(* Logix 5000 project; controller Comas_L4 vendor 1 type 14 code 193 rev 30.11; software revision 30.02; part 5 of 12 *)

VAR_GLOBAL   (* controller tags *)
   Activation_Mode_Once : BOOL;
   Activation_Pompe : BOOL := 1;
   Activation_Rouleau : BOOL := 1;
   Activation_Synchro_Directe_Codeur : BOOL := 1;
   AOI_Badge : Badges_Acces := (Tempo_Logout_1 := 600000, Tempo_Logout_2 := 3600000, Tempo_Logout_3 := 3600000);
   AOI_Cam_Display_Horiz : AOI_CamDisplay_OCX_StdCAM := (Sts_EN := 1);
   AOI_Cam_Display_Verti : AOI_CamDisplay_OCX_StdCAM := (Sts_EN := 1);
   AOI_Pilotage_Codeur_Vitesse_Moy : Pilotage_Vitesse_Rapide_V4 := (Vitesse := 46.548676, Acc := 1000.0, Dec := 1000.0, Jerk := 25.0, Autorisation := 1, St_Vitesse := 1);
   Axe_Codeur_Four : AXIS_CIP_DRIVE;
   Axe_Comas : MOTION_GROUP;
   Axe_Coupe_Fil : AXIS_CIP_DRIVE;
   Axe_Horizontal_Droit : AXIS_CIP_DRIVE;
   Axe_Horizontal_Gauche : AXIS_CIP_DRIVE;
   Axe_Pompe_Doseuse : AXIS_CIP_DRIVE;
   Axe_Rouleaux_Canneles : AXIS_CIP_DRIVE;
   Axe_Vertical_Droit : AXIS_CIP_DRIVE;
   Axe_Vertical_Gauche : AXIS_CIP_DRIVE;
   Axe_Virtuel_Codeur : AXIS_VIRTUAL;
   Axe_Virtuel_Codeur_test : AXIS_VIRTUAL;
   Axe_Virtuel_Coupe_Fil : AXIS_VIRTUAL;
   Axe_Virtuel_Maitre : AXIS_VIRTUAL;
   Badge_Code_A : BOOL;
   Badge_Code_B : BOOL;
   Badge_Code_C : BOOL;
   Badge_Code_D : BOOL;
   BP_O_F_Trappe : BOOL;
   Cadencement_Moyennage_Codeur : FBD_TIMER := (TimerEnable := 1, PRE := 1000, ACC := 930, EN := 1, TT := 1);
   Cam_Chart_Horiz : Chart := (NumberOfDataPoints := 130, X_Axis_Min := -1.0, X_Axis_Max := 90.0, Y_Axis_Min := -52.012157, Y_Axis_Max := 87.0, DataSeries_FixedAxis.Visible := 1, DataSeries_FixedAxis.Data[1] := 0.6923077, DataSeries_FixedAxis.Data[2] := 1.3846154, DataSeries_FixedAxis.Data[3] := 2.0769231, DataSeries_FixedAxis.Data[4] := 2.7692308, DataSeries_FixedAxis.Data[5] := 3.4615386, DataSeries_FixedAxis.Data[6] := 4.1538463, DataSeries_FixedAxis.Data[7] := 4.846154, DataSeries_FixedAxis.Data[8] := 5.5384617, DataSeries_FixedAxis.Data[9] := 6.230769, DataSeries_FixedAxis.Data[10] := 6.9230766, DataSeries_FixedAxis.Data[11] := 7.615384, DataSeries_FixedAxis.Data[12] := 8.307692, DataSeries_FixedAxis.Data[13] := 8.999999, DataSeries_FixedAxis.Data[14] := 9.6923065, DataSeries_FixedAxis.Data[15] := 10.384614, DataSeries_FixedAxis.Data[16] := 11.076921, DataSeries_FixedAxis.Data[17] := 11.769229, DataSeries_FixedAxis.Data[18] := 12.461536, DataSeries_FixedAxis.Data[19] := 13.153844, DataSeries_FixedAxis.Data[20] := 13.846151, DataSeries_FixedAxis.Data[21] := 14.538459, DataSeries_FixedAxis.Data[22] := 15.230766, DataSeries_FixedAxis.Data[23] := 15.923074, DataSeries_FixedAxis.Data[24] := 16.615381, DataSeries_FixedAxis.Data[25] := 17.30769, DataSeries_FixedAxis.Data[26] := 17.999998, DataSeries_FixedAxis.Data[27] := 18.692307, DataSeries_FixedAxis.Data[28] := 19.384615, DataSeries_FixedAxis.Data[29] := 20.076923, DataSeries_FixedAxis.Data[30] := 20.769232, DataSeries_FixedAxis.Data[31] := 21.46154, DataSeries_FixedAxis.Data[32] := 22.153849, DataSeries_FixedAxis.Data[33] := 22.846157, DataSeries_FixedAxis.Data[34] := 23.538465, DataSeries_FixedAxis.Data[35] := 24.230774, DataSeries_FixedAxis.Data[36] := 24.923082, DataSeries_FixedAxis.Data[37] := 25.61539, DataSeries_FixedAxis.Data[38] := 26.3077, DataSeries_FixedAxis.Data[39] := 27.000008, DataSeries_FixedAxis.Data[40] := 27.692316, DataSeries_FixedAxis.Data[41] := 28.384624, DataSeries_FixedAxis.Data[42] := 29.076933, DataSeries_FixedAxis.Data[43] := 29.769241, DataSeries_FixedAxis.Data[44] := 30.46155, DataSeries_FixedAxis.Data[45] := 31.153858, DataSeries_FixedAxis.Data[46] := 31.846167, DataSeries_FixedAxis.Data[47] := 32.538475, DataSeries_FixedAxis.Data[48] := 33.23078, DataSeries_FixedAxis.Data[49] := 33.923088, DataSeries_FixedAxis.Data[50] := 34.615395, DataSeries_FixedAxis.Data[51] := 35.3077, DataSeries_FixedAxis.Data[52] := 36.000008, DataSeries_FixedAxis.Data[53] := 36.692314, DataSeries_FixedAxis.Data[54] := 37.38462,
        DataSeries_FixedAxis.Data[55] := 38.076927, DataSeries_FixedAxis.Data[56] := 38.769234, DataSeries_FixedAxis.Data[57] := 39.46154, DataSeries_FixedAxis.Data[58] := 40.153847, DataSeries_FixedAxis.Data[59] := 40.846153, DataSeries_FixedAxis.Data[60] := 41.53846, DataSeries_FixedAxis.Data[61] := 42.230766, DataSeries_FixedAxis.Data[62] := 42.923073, DataSeries_FixedAxis.Data[63] := 43.61538, DataSeries_FixedAxis.Data[64] := 44.307686, DataSeries_FixedAxis.Data[65] := 44.999992, DataSeries_FixedAxis.Data[66] := 45.6923, DataSeries_FixedAxis.Data[67] := 46.384605, DataSeries_FixedAxis.Data[68] := 47.076912, DataSeries_FixedAxis.Data[69] := 47.76922, DataSeries_FixedAxis.Data[70] := 48.461525, DataSeries_FixedAxis.Data[71] := 49.15383, DataSeries_FixedAxis.Data[72] := 49.846138, DataSeries_FixedAxis.Data[73] := 50.538445, DataSeries_FixedAxis.Data[74] := 51.23075, DataSeries_FixedAxis.Data[75] := 51.923058, DataSeries_FixedAxis.Data[76] := 52.615364, DataSeries_FixedAxis.Data[77] := 53.30767, DataSeries_FixedAxis.Data[78] := 53.999977, DataSeries_FixedAxis.Data[79] := 54.692284, DataSeries_FixedAxis.Data[80] := 55.38459, DataSeries_FixedAxis.Data[81] := 56.076897, DataSeries_FixedAxis.Data[82] := 56.769203, DataSeries_FixedAxis.Data[83] := 57.46151, DataSeries_FixedAxis.Data[84] := 58.153816, DataSeries_FixedAxis.Data[85] := 58.846123, DataSeries_FixedAxis.Data[86] := 59.53843, DataSeries_FixedAxis.Data[87] := 60.230736, DataSeries_FixedAxis.Data[88] := 60.923042, DataSeries_FixedAxis.Data[89] := 61.61535, DataSeries_FixedAxis.Data[90] := 62.307655, DataSeries_FixedAxis.Data[91] := 62.99996, DataSeries_FixedAxis.Data[92] := 63.69227, DataSeries_FixedAxis.Data[93] := 64.384575, DataSeries_FixedAxis.Data[94] := 65.07688, DataSeries_FixedAxis.Data[95] := 65.76919, DataSeries_FixedAxis.Data[96] := 66.461494, DataSeries_FixedAxis.Data[97] := 67.1538, DataSeries_FixedAxis.Data[98] := 67.84611, DataSeries_FixedAxis.Data[99] := 68.538414, DataSeries_FixedAxis.Data[100] := 69.23072, DataSeries_FixedAxis.Data[101] := 69.92303, DataSeries_FixedAxis.Data[102] := 70.61533, DataSeries_FixedAxis.Data[103] := 71.30764, DataSeries_FixedAxis.Data[104] := 71.99995, DataSeries_FixedAxis.Data[105] := 72.69225, DataSeries_FixedAxis.Data[106] := 73.38456, DataSeries_FixedAxis.Data[107] := 74.076866, DataSeries_FixedAxis.Data[108] := 74.76917, DataSeries_FixedAxis.Data[109] := 75.46148, DataSeries_FixedAxis.Data[110] := 76.153786, DataSeries_FixedAxis.Data[111] := 76.84609, DataSeries_FixedAxis.Data[112] := 77.5384, DataSeries_FixedAxis.Data[113] := 78.230705, DataSeries_FixedAxis.Data[114] := 78.92301,
        DataSeries_FixedAxis.Data[115] := 79.61532, DataSeries_FixedAxis.Data[116] := 80.307625, DataSeries_FixedAxis.Data[117] := 80.99993, DataSeries_FixedAxis.Data[118] := 81.69224, DataSeries_FixedAxis.Data[119] := 82.384544, DataSeries_FixedAxis.Data[120] := 83.07685, DataSeries_FixedAxis.Data[121] := 83.76916, DataSeries_FixedAxis.Data[122] := 84.461464, DataSeries_FixedAxis.Data[123] := 85.15377, DataSeries_FixedAxis.Data[124] := 85.84608, DataSeries_FixedAxis.Data[125] := 86.53838, DataSeries_FixedAxis.Data[126] := 87.23069, DataSeries_FixedAxis.Data[127] := 87.923, DataSeries_FixedAxis.Data[128] := 88.6153, DataSeries_FixedAxis.Data[129] := 90.0, DataSeries_1.Label := 'Position', DataSeries_1.Visible := 1, DataSeries_1.Data[2] := 0.018661816, DataSeries_1.Data[3] := 0.15915523, DataSeries_1.Data[4] := 0.46422943, DataSeries_1.Data[5] := 0.96573883, DataSeries_1.Data[6] := 1.6955377, DataSeries_1.Data[7] := 2.6854808, DataSeries_1.Data[8] := 3.9674213, DataSeries_1.Data[9] := 5.553846, DataSeries_1.Data[10] := 7.215384, DataSeries_1.Data[11] := 8.876922, DataSeries_1.Data[12] := 10.53846, DataSeries_1.Data[13] := 12.199998, DataSeries_1.Data[14] := 13.861536, DataSeries_1.Data[15] := 15.523073, DataSeries_1.Data[16] := 17.184612, DataSeries_1.Data[17] := 18.84615, DataSeries_1.Data[18] := 20.507687, DataSeries_1.Data[19] := 22.169226, DataSeries_1.Data[20] := 23.830763, DataSeries_1.Data[21] := 25.492302, DataSeries_1.Data[22] := 27.15384, DataSeries_1.Data[23] := 28.815376, DataSeries_1.Data[24] := 30.476915, DataSeries_1.Data[25] := 32.138454, DataSeries_1.Data[26] := 33.799995, DataSeries_1.Data[27] := 35.461536, DataSeries_1.Data[28] := 37.123077, DataSeries_1.Data[29] := 38.784615, DataSeries_1.Data[30] := 40.446156, DataSeries_1.Data[31] := 42.107697, DataSeries_1.Data[32] := 43.769238, DataSeries_1.Data[33] := 45.43078, DataSeries_1.Data[34] := 47.092316, DataSeries_1.Data[35] := 48.753857, DataSeries_1.Data[36] := 50.415398, DataSeries_1.Data[37] := 52.07694, DataSeries_1.Data[38] := 53.73848, DataSeries_1.Data[39] := 55.400017, DataSeries_1.Data[40] := 57.061558, DataSeries_1.Data[41] := 58.7231, DataSeries_1.Data[42] := 60.38464, DataSeries_1.Data[43] := 62.04618, DataSeries_1.Data[44] := 63.707718,
        DataSeries_1.Data[45] := 65.36926, DataSeries_1.Data[46] := 67.0308, DataSeries_1.Data[47] := 68.69234, DataSeries_1.Data[48] := 70.353874, DataSeries_1.Data[49] := 72.01541, DataSeries_1.Data[50] := 73.67695, DataSeries_1.Data[51] := 75.338486, DataSeries_1.Data[52] := 77.000015, DataSeries_1.Data[53] := 78.57661, DataSeries_1.Data[54] := 79.98862, DataSeries_1.Data[55] := 81.24401, DataSeries_1.Data[56] := 82.350746, DataSeries_1.Data[57] := 83.316795, DataSeries_1.Data[58] := 84.15012, DataSeries_1.Data[59] := 84.85868, DataSeries_1.Data[60] := 85.45045, DataSeries_1.Data[61] := 85.93337, DataSeries_1.Data[62] := 86.31543, DataSeries_1.Data[63] := 86.604576, DataSeries_1.Data[64] := 86.80878, DataSeries_1.Data[65] := 86.936, DataSeries_1.Data[66] := 86.9942, DataSeries_1.Data[67] := 87.0, DataSeries_1.Data[68] := 87.0, DataSeries_1.Data[69] := 87.0, DataSeries_1.Data[70] := 87.0, DataSeries_1.Data[71] := 87.0, DataSeries_1.Data[72] := 87.0, DataSeries_1.Data[73] := 87.0, DataSeries_1.Data[74] := 86.995384, DataSeries_1.Data[75] := 86.92536, DataSeries_1.Data[76] := 86.76894, DataSeries_1.Data[77] := 86.52342, DataSeries_1.Data[78] := 86.18607, DataSeries_1.Data[79] := 85.75417, DataSeries_1.Data[80] := 85.225006, DataSeries_1.Data[81] := 84.595856, DataSeries_1.Data[82] := 83.86399, DataSeries_1.Data[83] := 83.0267, DataSeries_1.Data[84] := 82.08127, DataSeries_1.Data[85] := 81.02497, DataSeries_1.Data[86] := 79.85508, DataSeries_1.Data[87] := 78.56889, DataSeries_1.Data[88] := 77.16367, DataSeries_1.Data[89] := 75.63791, DataSeries_1.Data[90] := 73.99678, DataSeries_1.Data[91] := 72.247795, DataSeries_1.Data[92] := 70.39847, DataSeries_1.Data[93] := 68.45631, DataSeries_1.Data[94] := 66.42883, DataSeries_1.Data[95] := 64.323555, DataSeries_1.Data[96] := 62.14799, DataSeries_1.Data[97] := 59.90965, DataSeries_1.Data[98] := 57.61604, DataSeries_1.Data[99] := 55.27468, DataSeries_1.Data[100] := 52.893085, DataSeries_1.Data[101] := 50.478764, DataSeries_1.Data[102] := 48.039234, DataSeries_1.Data[103] := 45.582005, DataSeries_1.Data[104] := 43.11459,
        DataSeries_1.Data[105] := 40.644505, DataSeries_1.Data[106] := 38.17926, DataSeries_1.Data[107] := 35.726368, DataSeries_1.Data[108] := 33.293346, DataSeries_1.Data[109] := 30.887705, DataSeries_1.Data[110] := 28.516958, DataSeries_1.Data[111] := 26.188618, DataSeries_1.Data[112] := 23.910198, DataSeries_1.Data[113] := 21.68921, DataSeries_1.Data[114] := 19.53317, DataSeries_1.Data[115] := 17.44959, DataSeries_1.Data[116] := 15.445984, DataSeries_1.Data[117] := 13.529863, DataSeries_1.Data[118] := 11.708741, DataSeries_1.Data[119] := 9.990131, DataSeries_1.Data[120] := 8.381547, DataSeries_1.Data[121] := 6.890502, DataSeries_1.Data[122] := 5.524508, DataSeries_1.Data[123] := 4.2910795, DataSeries_1.Data[124] := 3.1977286, DataSeries_1.Data[125] := 2.251969, DataSeries_1.Data[126] := 1.461314, DataSeries_1.Data[127] := 0.83327633, DataSeries_1.Data[128] := 0.37536937, DataSeries_2.Label := 'Velocity', DataSeries_2.Visible := 1, DataSeries_2.Data[2] := 1.4492007, DataSeries_2.Data[3] := 4.579474, DataSeries_2.Data[4] := 8.38052, DataSeries_2.Data[5] := 12.85234, DataSeries_2.Data[6] := 17.994932, DataSeries_2.Data[7] := 23.808298, DataSeries_2.Data[8] := 30.292437, DataSeries_2.Data[9] := 34.987846, DataSeries_2.Data[10] := 34.987846, DataSeries_2.Data[11] := 34.987846, DataSeries_2.Data[12] := 34.987846, DataSeries_2.Data[13] := 34.987846, DataSeries_2.Data[14] := 34.987846, DataSeries_2.Data[15] := 34.987846, DataSeries_2.Data[16] := 34.987846, DataSeries_2.Data[17] := 34.987846, DataSeries_2.Data[18] := 34.987846, DataSeries_2.Data[19] := 34.987846, DataSeries_2.Data[20] := 34.987846, DataSeries_2.Data[21] := 34.987846, DataSeries_2.Data[22] := 34.987846, DataSeries_2.Data[23] := 34.987846, DataSeries_2.Data[24] := 34.987846, DataSeries_2.Data[25] := 34.987846, DataSeries_2.Data[26] := 34.987846, DataSeries_2.Data[27] := 34.987846, DataSeries_2.Data[28] := 34.987846, DataSeries_2.Data[29] := 34.987846, DataSeries_2.Data[30] := 34.987846, DataSeries_2.Data[31] := 34.987846, DataSeries_2.Data[32] := 34.987846, DataSeries_2.Data[33] := 34.987846, DataSeries_2.Data[34] := 34.987846, DataSeries_2.Data[35] := 34.987846,
        DataSeries_2.Data[36] := 34.987846, DataSeries_2.Data[37] := 34.987846, DataSeries_2.Data[38] := 34.987846, DataSeries_2.Data[39] := 34.987846, DataSeries_2.Data[40] := 34.987846, DataSeries_2.Data[41] := 34.987846, DataSeries_2.Data[42] := 34.987846, DataSeries_2.Data[43] := 34.987846, DataSeries_2.Data[44] := 34.987846, DataSeries_2.Data[45] := 34.987846, DataSeries_2.Data[46] := 34.987846, DataSeries_2.Data[47] := 34.987846, DataSeries_2.Data[48] := 34.987846, DataSeries_2.Data[49] := 34.987846, DataSeries_2.Data[50] := 34.987846, DataSeries_2.Data[51] := 34.987846, DataSeries_2.Data[52] := 34.987804, DataSeries_2.Data[53] := 31.438305, DataSeries_2.Data[54] := 28.0565, DataSeries_2.Data[55] := 24.842386, DataSeries_2.Data[56] := 21.795965, DataSeries_2.Data[57] := 18.917236, DataSeries_2.Data[58] := 16.206202, DataSeries_2.Data[59] := 13.662858, DataSeries_2.Data[60] := 11.287208, DataSeries_2.Data[61] := 9.07925, DataSeries_2.Data[62] := 7.038986, DataSeries_2.Data[63] := 5.166414, DataSeries_2.Data[64] := 3.4615343, DataSeries_2.Data[65] := 1.9243474, DataSeries_2.Data[66] := 0.55485314, DataSeries_2.Data[74] := -0.58406484, DataSeries_2.Data[75] := -2.3745732, DataSeries_2.Data[76] := -4.2223506, DataSeries_2.Data[77] := -6.1273975, DataSeries_2.Data[78] := -8.089713, DataSeries_2.Data[79] := -10.109298, DataSeries_2.Data[80] := -12.186151, DataSeries_2.Data[81] := -14.320274, DataSeries_2.Data[82] := -16.511665, DataSeries_2.Data[83] := -18.760324, DataSeries_2.Data[84] := -21.066257, DataSeries_2.Data[85] := -23.429455, DataSeries_2.Data[86] := -25.849922, DataSeries_2.Data[87] := -28.32766, DataSeries_2.Data[88] := -30.862663, DataSeries_2.Data[89] := -33.369823, DataSeries_2.Data[90] := -35.720104, DataSeries_2.Data[91] := -37.912178, DataSeries_2.Data[92] := -39.94604, DataSeries_2.Data[93] := -41.821697, DataSeries_2.Data[94] := -43.539146, DataSeries_2.Data[95] := -45.09838, DataSeries_2.Data[96] := -46.499413, DataSeries_2.Data[97] := -47.742233, DataSeries_2.Data[98] := -48.82685, DataSeries_2.Data[99] := -49.753258, DataSeries_2.Data[100] := -50.52145, DataSeries_2.Data[101] := -51.131443, DataSeries_2.Data[102] := -51.58322,
        DataSeries_2.Data[103] := -51.876797, DataSeries_2.Data[104] := -52.012157, DataSeries_2.Data[105] := -51.989315, DataSeries_2.Data[106] := -51.80826, DataSeries_2.Data[107] := -51.468998, DataSeries_2.Data[108] := -50.97153, DataSeries_2.Data[109] := -50.315853, DataSeries_2.Data[110] := -49.50197, DataSeries_2.Data[111] := -48.529873, DataSeries_2.Data[112] := -47.39957, DataSeries_2.Data[113] := -46.111057, DataSeries_2.Data[114] := -44.66434, DataSeries_2.Data[115] := -43.05941, DataSeries_2.Data[116] := -41.296272, DataSeries_2.Data[117] := -39.374928, DataSeries_2.Data[118] := -37.29538, DataSeries_2.Data[119] := -35.057617, DataSeries_2.Data[120] := -32.661648, DataSeries_2.Data[121] := -30.107468, DataSeries_2.Data[122] := -27.39508, DataSeries_2.Data[123] := -24.524488, DataSeries_2.Data[124] := -21.495686, DataSeries_2.Data[125] := -18.308674, DataSeries_2.Data[126] := -14.963453, DataSeries_2.Data[127] := -11.460026, DataSeries_2.Data[128] := -7.7983894, DataSeries_3.Label := 'Acceleration', DataSeries_3.Visible := 1, DataSeries_3.Data[2] := 23.262037, DataSeries_3.Data[3] := 28.844927, DataSeries_3.Data[4] := 34.427814, DataSeries_3.Data[5] := 40.010704, DataSeries_3.Data[6] := 45.593594, DataSeries_3.Data[7] := 51.176487, DataSeries_3.Data[8] := 56.759373, DataSeries_3.Data[52] := -30.240631, DataSeries_3.Data[53] := -28.844913, DataSeries_3.Data[54] := -27.449194, DataSeries_3.Data[55] := -26.053474, DataSeries_3.Data[56] := -24.657753, DataSeries_3.Data[57] := -23.262033, DataSeries_3.Data[58] := -21.866312, DataSeries_3.Data[59] := -20.470594, DataSeries_3.Data[60] := -19.074873, DataSeries_3.Data[61] := -17.679153, DataSeries_3.Data[62] := -16.283434, DataSeries_3.Data[63] := -14.887714, DataSeries_3.Data[64] := -13.491994, DataSeries_3.Data[65] := -12.096275, DataSeries_3.Data[66] := -10.700555, DataSeries_3.Data[74] := -14.664224, DataSeries_3.Data[75] := -15.140878, DataSeries_3.Data[76] := -15.617534, DataSeries_3.Data[77] := -16.094189, DataSeries_3.Data[78] := -16.570843, DataSeries_3.Data[79] := -17.047499, DataSeries_3.Data[80] := -17.524153, DataSeries_3.Data[81] := -18.000809, DataSeries_3.Data[82] := -18.477463, DataSeries_3.Data[83] := -18.954119,
        DataSeries_3.Data[84] := -19.430773, DataSeries_3.Data[85] := -19.907429, DataSeries_3.Data[86] := -20.384083, DataSeries_3.Data[87] := -20.860739, DataSeries_3.Data[88] := -21.337395, DataSeries_3.Data[89] := -20.219973, DataSeries_3.Data[90] := -18.903193, DataSeries_3.Data[91] := -17.58641, DataSeries_3.Data[92] := -16.269629, DataSeries_3.Data[93] := -14.9528475, DataSeries_3.Data[94] := -13.636066, DataSeries_3.Data[95] := -12.319286, DataSeries_3.Data[96] := -11.002504, DataSeries_3.Data[97] := -9.685723, DataSeries_3.Data[98] := -8.368942, DataSeries_3.Data[99] := -7.0521607, DataSeries_3.Data[100] := -5.735379, DataSeries_3.Data[101] := -4.418598, DataSeries_3.Data[102] := -3.1018171, DataSeries_3.Data[103] := -1.7850357, DataSeries_3.Data[104] := -0.46825457, DataSeries_3.Data[105] := 0.84852666, DataSeries_3.Data[106] := 2.165308, DataSeries_3.Data[107] := 3.482089, DataSeries_3.Data[108] := 4.79887, DataSeries_3.Data[109] := 6.1156516, DataSeries_3.Data[110] := 7.4324327, DataSeries_3.Data[111] := 8.749214, DataSeries_3.Data[112] := 10.065995, DataSeries_3.Data[113] := 11.382776, DataSeries_3.Data[114] := 12.699557, DataSeries_3.Data[115] := 14.016339, DataSeries_3.Data[116] := 15.33312, DataSeries_3.Data[117] := 16.649902, DataSeries_3.Data[118] := 17.966682, DataSeries_3.Data[119] := 19.283464, DataSeries_3.Data[120] := 20.600245, DataSeries_3.Data[121] := 21.917025, DataSeries_3.Data[122] := 23.233807, DataSeries_3.Data[123] := 24.550589, DataSeries_3.Data[124] := 25.86737, DataSeries_3.Data[125] := 27.18415, DataSeries_3.Data[126] := 28.500933, DataSeries_3.Data[127] := 29.817715, DataSeries_3.Data[128] := 31.134497);
   Cam_Chart_Verti : Chart := (NumberOfDataPoints := 130, X_Axis_Max := 90.0, Y_Axis_Min := -4.9572415, Y_Axis_Max := 25.0, DataSeries_FixedAxis.Visible := 1, DataSeries_FixedAxis.Data[1] := 0.6923077, DataSeries_FixedAxis.Data[2] := 1.3846154, DataSeries_FixedAxis.Data[3] := 2.0769231, DataSeries_FixedAxis.Data[4] := 2.7692308, DataSeries_FixedAxis.Data[5] := 3.4615386, DataSeries_FixedAxis.Data[6] := 4.1538463, DataSeries_FixedAxis.Data[7] := 4.846154, DataSeries_FixedAxis.Data[8] := 5.5384617, DataSeries_FixedAxis.Data[9] := 6.230769, DataSeries_FixedAxis.Data[10] := 6.9230766, DataSeries_FixedAxis.Data[11] := 7.615384, DataSeries_FixedAxis.Data[12] := 8.307692, DataSeries_FixedAxis.Data[13] := 8.999999, DataSeries_FixedAxis.Data[14] := 9.6923065, DataSeries_FixedAxis.Data[15] := 10.384614, DataSeries_FixedAxis.Data[16] := 11.076921, DataSeries_FixedAxis.Data[17] := 11.769229, DataSeries_FixedAxis.Data[18] := 12.461536, DataSeries_FixedAxis.Data[19] := 13.153844, DataSeries_FixedAxis.Data[20] := 13.846151, DataSeries_FixedAxis.Data[21] := 14.538459, DataSeries_FixedAxis.Data[22] := 15.230766, DataSeries_FixedAxis.Data[23] := 15.923074, DataSeries_FixedAxis.Data[24] := 16.615381, DataSeries_FixedAxis.Data[25] := 17.30769, DataSeries_FixedAxis.Data[26] := 17.999998, DataSeries_FixedAxis.Data[27] := 18.692307, DataSeries_FixedAxis.Data[28] := 19.384615, DataSeries_FixedAxis.Data[29] := 20.076923, DataSeries_FixedAxis.Data[30] := 20.769232, DataSeries_FixedAxis.Data[31] := 21.46154, DataSeries_FixedAxis.Data[32] := 22.153849, DataSeries_FixedAxis.Data[33] := 22.846157, DataSeries_FixedAxis.Data[34] := 23.538465, DataSeries_FixedAxis.Data[35] := 24.230774, DataSeries_FixedAxis.Data[36] := 24.923082, DataSeries_FixedAxis.Data[37] := 25.61539, DataSeries_FixedAxis.Data[38] := 26.3077, DataSeries_FixedAxis.Data[39] := 27.000008, DataSeries_FixedAxis.Data[40] := 27.692316, DataSeries_FixedAxis.Data[41] := 28.384624, DataSeries_FixedAxis.Data[42] := 29.076933, DataSeries_FixedAxis.Data[43] := 29.769241, DataSeries_FixedAxis.Data[44] := 30.46155, DataSeries_FixedAxis.Data[45] := 31.153858, DataSeries_FixedAxis.Data[46] := 31.846167, DataSeries_FixedAxis.Data[47] := 32.538475, DataSeries_FixedAxis.Data[48] := 33.23078, DataSeries_FixedAxis.Data[49] := 33.923088, DataSeries_FixedAxis.Data[50] := 34.615395, DataSeries_FixedAxis.Data[51] := 35.3077, DataSeries_FixedAxis.Data[52] := 36.000008, DataSeries_FixedAxis.Data[53] := 36.692314, DataSeries_FixedAxis.Data[54] := 37.38462, DataSeries_FixedAxis.Data[55] := 38.076927,
        DataSeries_FixedAxis.Data[56] := 38.769234, DataSeries_FixedAxis.Data[57] := 39.46154, DataSeries_FixedAxis.Data[58] := 40.153847, DataSeries_FixedAxis.Data[59] := 40.846153, DataSeries_FixedAxis.Data[60] := 41.53846, DataSeries_FixedAxis.Data[61] := 42.230766, DataSeries_FixedAxis.Data[62] := 42.923073, DataSeries_FixedAxis.Data[63] := 43.61538, DataSeries_FixedAxis.Data[64] := 44.307686, DataSeries_FixedAxis.Data[65] := 44.999992, DataSeries_FixedAxis.Data[66] := 45.6923, DataSeries_FixedAxis.Data[67] := 46.384605, DataSeries_FixedAxis.Data[68] := 47.076912, DataSeries_FixedAxis.Data[69] := 47.76922, DataSeries_FixedAxis.Data[70] := 48.461525, DataSeries_FixedAxis.Data[71] := 49.15383, DataSeries_FixedAxis.Data[72] := 49.846138, DataSeries_FixedAxis.Data[73] := 50.538445, DataSeries_FixedAxis.Data[74] := 51.23075, DataSeries_FixedAxis.Data[75] := 51.923058, DataSeries_FixedAxis.Data[76] := 52.615364, DataSeries_FixedAxis.Data[77] := 53.30767, DataSeries_FixedAxis.Data[78] := 53.999977, DataSeries_FixedAxis.Data[79] := 54.692284, DataSeries_FixedAxis.Data[80] := 55.38459, DataSeries_FixedAxis.Data[81] := 56.076897, DataSeries_FixedAxis.Data[82] := 56.769203, DataSeries_FixedAxis.Data[83] := 57.46151, DataSeries_FixedAxis.Data[84] := 58.153816, DataSeries_FixedAxis.Data[85] := 58.846123, DataSeries_FixedAxis.Data[86] := 59.53843, DataSeries_FixedAxis.Data[87] := 60.230736, DataSeries_FixedAxis.Data[88] := 60.923042, DataSeries_FixedAxis.Data[89] := 61.61535, DataSeries_FixedAxis.Data[90] := 62.307655, DataSeries_FixedAxis.Data[91] := 62.99996, DataSeries_FixedAxis.Data[92] := 63.69227, DataSeries_FixedAxis.Data[93] := 64.384575, DataSeries_FixedAxis.Data[94] := 65.07688, DataSeries_FixedAxis.Data[95] := 65.76919, DataSeries_FixedAxis.Data[96] := 66.461494, DataSeries_FixedAxis.Data[97] := 67.1538, DataSeries_FixedAxis.Data[98] := 67.84611, DataSeries_FixedAxis.Data[99] := 68.538414, DataSeries_FixedAxis.Data[100] := 69.23072, DataSeries_FixedAxis.Data[101] := 69.92303, DataSeries_FixedAxis.Data[102] := 70.61533, DataSeries_FixedAxis.Data[103] := 71.30764, DataSeries_FixedAxis.Data[104] := 71.99995, DataSeries_FixedAxis.Data[105] := 72.69225, DataSeries_FixedAxis.Data[106] := 73.38456, DataSeries_FixedAxis.Data[107] := 74.076866, DataSeries_FixedAxis.Data[108] := 74.76917, DataSeries_FixedAxis.Data[109] := 75.46148, DataSeries_FixedAxis.Data[110] := 76.153786, DataSeries_FixedAxis.Data[111] := 76.84609, DataSeries_FixedAxis.Data[112] := 77.5384, DataSeries_FixedAxis.Data[113] := 78.230705, DataSeries_FixedAxis.Data[114] := 78.92301, DataSeries_FixedAxis.Data[115] := 79.61532,
        DataSeries_FixedAxis.Data[116] := 80.307625, DataSeries_FixedAxis.Data[117] := 80.99993, DataSeries_FixedAxis.Data[118] := 81.69224, DataSeries_FixedAxis.Data[119] := 82.384544, DataSeries_FixedAxis.Data[120] := 83.07685, DataSeries_FixedAxis.Data[121] := 83.76916, DataSeries_FixedAxis.Data[122] := 84.461464, DataSeries_FixedAxis.Data[123] := 85.15377, DataSeries_FixedAxis.Data[124] := 85.84608, DataSeries_FixedAxis.Data[125] := 86.53838, DataSeries_FixedAxis.Data[126] := 87.23069, DataSeries_FixedAxis.Data[127] := 87.923, DataSeries_FixedAxis.Data[128] := 88.6153, DataSeries_FixedAxis.Data[129] := 90.0, DataSeries_1.Label := 'Position', DataSeries_1.Visible := 1, DataSeries_1.Data[0] := 15.0, DataSeries_1.Data[1] := 15.0, DataSeries_1.Data[2] := 15.0, DataSeries_1.Data[3] := 15.0, DataSeries_1.Data[4] := 15.0, DataSeries_1.Data[5] := 15.0, DataSeries_1.Data[6] := 15.0, DataSeries_1.Data[7] := 15.0, DataSeries_1.Data[8] := 15.0, DataSeries_1.Data[9] := 15.0, DataSeries_1.Data[10] := 15.0, DataSeries_1.Data[11] := 15.0, DataSeries_1.Data[12] := 15.0, DataSeries_1.Data[13] := 15.0, DataSeries_1.Data[14] := 15.0, DataSeries_1.Data[15] := 15.0, DataSeries_1.Data[16] := 15.0, DataSeries_1.Data[17] := 15.0, DataSeries_1.Data[18] := 15.0, DataSeries_1.Data[19] := 15.0, DataSeries_1.Data[20] := 15.0, DataSeries_1.Data[21] := 15.0, DataSeries_1.Data[22] := 15.0, DataSeries_1.Data[23] := 15.0, DataSeries_1.Data[24] := 15.0, DataSeries_1.Data[25] := 15.0, DataSeries_1.Data[26] := 15.0, DataSeries_1.Data[27] := 15.0, DataSeries_1.Data[28] := 15.0, DataSeries_1.Data[29] := 15.0, DataSeries_1.Data[30] := 15.0, DataSeries_1.Data[31] := 15.0, DataSeries_1.Data[32] := 15.0, DataSeries_1.Data[33] := 15.0, DataSeries_1.Data[34] := 15.0, DataSeries_1.Data[35] := 15.0, DataSeries_1.Data[36] := 15.0, DataSeries_1.Data[37] := 15.0, DataSeries_1.Data[38] := 15.0, DataSeries_1.Data[39] := 15.0, DataSeries_1.Data[40] := 15.0, DataSeries_1.Data[41] := 15.0, DataSeries_1.Data[42] := 15.0, DataSeries_1.Data[43] := 15.0,
        DataSeries_1.Data[44] := 15.0, DataSeries_1.Data[45] := 15.0, DataSeries_1.Data[46] := 15.0, DataSeries_1.Data[47] := 15.0, DataSeries_1.Data[48] := 15.0, DataSeries_1.Data[49] := 15.0, DataSeries_1.Data[50] := 15.0, DataSeries_1.Data[51] := 15.0, DataSeries_1.Data[52] := 15.0, DataSeries_1.Data[53] := 15.0, DataSeries_1.Data[54] := 15.0, DataSeries_1.Data[55] := 15.0, DataSeries_1.Data[56] := 15.0, DataSeries_1.Data[57] := 15.0, DataSeries_1.Data[58] := 15.0, DataSeries_1.Data[59] := 15.0, DataSeries_1.Data[60] := 15.0, DataSeries_1.Data[61] := 15.0, DataSeries_1.Data[62] := 15.0, DataSeries_1.Data[63] := 15.0, DataSeries_1.Data[64] := 15.0, DataSeries_1.Data[65] := 15.0, DataSeries_1.Data[66] := 15.0, DataSeries_1.Data[67] := 15.0, DataSeries_1.Data[68] := 15.0, DataSeries_1.Data[69] := 15.0, DataSeries_1.Data[70] := 15.061935, DataSeries_1.Data[71] := 15.368675, DataSeries_1.Data[72] := 15.896626, DataSeries_1.Data[73] := 16.60597, DataSeries_1.Data[74] := 17.45689, DataSeries_1.Data[75] := 18.409567, DataSeries_1.Data[76] := 19.424185, DataSeries_1.Data[77] := 20.460924, DataSeries_1.Data[78] := 21.479967, DataSeries_1.Data[79] := 22.441498, DataSeries_1.Data[80] := 23.305696, DataSeries_1.Data[81] := 24.032747, DataSeries_1.Data[82] := 24.582832, DataSeries_1.Data[83] := 24.916132, DataSeries_1.Data[84] := 25.0, DataSeries_1.Data[85] := 25.0, DataSeries_1.Data[86] := 25.0, DataSeries_1.Data[87] := 25.0, DataSeries_1.Data[88] := 25.0, DataSeries_1.Data[89] := 25.0, DataSeries_1.Data[90] := 25.0, DataSeries_1.Data[91] := 25.0, DataSeries_1.Data[92] := 24.956764, DataSeries_1.Data[93] := 24.831598, DataSeries_1.Data[94] := 24.63133, DataSeries_1.Data[95] := 24.362785, DataSeries_1.Data[96] := 24.032795, DataSeries_1.Data[97] := 23.648184, DataSeries_1.Data[98] := 23.215778, DataSeries_1.Data[99] := 22.74241, DataSeries_1.Data[100] := 22.234903, DataSeries_1.Data[101] := 21.700085, DataSeries_1.Data[102] := 21.144785, DataSeries_1.Data[103] := 20.575829,
        DataSeries_1.Data[104] := 20.000044, DataSeries_1.Data[105] := 19.42426, DataSeries_1.Data[106] := 18.855303, DataSeries_1.Data[107] := 18.3, DataSeries_1.Data[108] := 17.765179, DataSeries_1.Data[109] := 17.257666, DataSeries_1.Data[110] := 16.78429, DataSeries_1.Data[111] := 16.35188, DataSeries_1.Data[112] := 15.96726, DataSeries_1.Data[113] := 15.63726, DataSeries_1.Data[114] := 15.368707, DataSeries_1.Data[115] := 15.168427, DataSeries_1.Data[116] := 15.043249, DataSeries_1.Data[117] := 15.0, DataSeries_1.Data[118] := 15.0, DataSeries_1.Data[119] := 15.0, DataSeries_1.Data[120] := 15.0, DataSeries_1.Data[121] := 15.0, DataSeries_1.Data[122] := 15.0, DataSeries_1.Data[123] := 15.0, DataSeries_1.Data[124] := 15.0, DataSeries_1.Data[125] := 15.0, DataSeries_1.Data[126] := 15.0, DataSeries_1.Data[127] := 15.0, DataSeries_1.Data[128] := 15.0, DataSeries_1.Data[129] := 15.0, DataSeries_2.Label := 'Velocity', DataSeries_2.Visible := 1, DataSeries_2.Data[70] := 1.1347679, DataSeries_2.Data[71] := 2.6310582, DataSeries_2.Data[72] := 3.880256, DataSeries_2.Data[73] := 4.8823614, DataSeries_2.Data[74] := 5.6373744, DataSeries_2.Data[75] := 6.145294, DataSeries_2.Data[76] := 6.4061217, DataSeries_2.Data[77] := 6.4198565, DataSeries_2.Data[78] := 6.186499, DataSeries_2.Data[79] := 5.7060485, DataSeries_2.Data[80] := 4.978506, DataSeries_2.Data[81] := 4.0038705, DataSeries_2.Data[82] := 2.7821426, DataSeries_2.Data[83] := 1.313322, DataSeries_2.Data[92] := -0.5295781, DataSeries_2.Data[93] := -1.016818, DataSeries_2.Data[94] := -1.4616897, DataSeries_2.Data[95] := -1.8641928, DataSeries_2.Data[96] := -2.2243276, DataSeries_2.Data[97] := -2.542094, DataSeries_2.Data[98] := -2.817492, DataSeries_2.Data[99] := -3.0505214, DataSeries_2.Data[100] := -3.2411828, DataSeries_2.Data[101] := -3.3894756, DataSeries_2.Data[102] := -3.4953997, DataSeries_2.Data[103] := -3.5589557, DataSeries_2.Data[104] := -3.580143, DataSeries_2.Data[105] := -3.558962, DataSeries_2.Data[106] := -3.4954126, DataSeries_2.Data[107] := -3.389495, DataSeries_2.Data[108] := -3.241209, DataSeries_2.Data[109] := -3.0505543,
        DataSeries_2.Data[110] := -2.8175313, DataSeries_2.Data[111] := -2.5421398, DataSeries_2.Data[112] := -2.2243798, DataSeries_2.Data[113] := -1.8642517, DataSeries_2.Data[114] := -1.461755, DataSeries_2.Data[115] := -1.01689, DataSeries_2.Data[116] := -0.5296565, DataSeries_2.Data[117] := -5.462844e-05, DataSeries_3.Label := 'Acceleration', DataSeries_3.Visible := 1, DataSeries_3.Data[70] := 5.042759, DataSeries_3.Data[71] := 4.273528, DataSeries_3.Data[72] := 3.5042973, DataSeries_3.Data[73] := 2.7350667, DataSeries_3.Data[74] := 1.9658357, DataSeries_3.Data[75] := 1.1966048, DataSeries_3.Data[76] := 0.42737398, DataSeries_3.Data[77] := -0.34185684, DataSeries_3.Data[78] := -1.1110877, DataSeries_3.Data[79] := -1.8803184, DataSeries_3.Data[80] := -2.6495492, DataSeries_3.Data[81] := -3.4187799, DataSeries_3.Data[82] := -4.188011, DataSeries_3.Data[83] := -4.9572415, DataSeries_3.Data[92] := -1.5827897, DataSeries_3.Data[93] := -1.4508914, DataSeries_3.Data[94] := -1.3189931, DataSeries_3.Data[95] := -1.1870948, DataSeries_3.Data[96] := -1.0551964, DataSeries_3.Data[97] := -0.9232982, DataSeries_3.Data[98] := -0.7913999, DataSeries_3.Data[99] := -0.6595017, DataSeries_3.Data[100] := -0.5276033, DataSeries_3.Data[101] := -0.395705, DataSeries_3.Data[102] := -0.26380676, DataSeries_3.Data[103] := -0.13190846, DataSeries_3.Data[104] := -1.017487e-05, DataSeries_3.Data[105] := 0.13188812, DataSeries_3.Data[106] := 0.2637864, DataSeries_3.Data[107] := 0.3956847, DataSeries_3.Data[108] := 0.527583, DataSeries_3.Data[109] := 0.6594813, DataSeries_3.Data[110] := 0.7913796, DataSeries_3.Data[111] := 0.92327785, DataSeries_3.Data[112] := 1.0551761, DataSeries_3.Data[113] := 1.1870744, DataSeries_3.Data[114] := 1.3189727, DataSeries_3.Data[115] := 1.4508709, DataSeries_3.Data[116] := 1.5827692, DataSeries_3.Data[117] := 1.7146676);
   Cam_Display_Horiz : UDT_Axis_Cam_Profil := (Cam[1].Master := 1.0, Cam[1].SegmentType := 1, Cam[2].Master := 6.0, Cam[2].Slave := 5.0, Cam[3].Master := 36.0, Cam[3].Slave := 77.0, Cam[3].SegmentType := 1, Cam[4].Master := 46.0, Cam[4].Slave := 87.0, Cam[5].Master := 51.0, Cam[5].Slave := 87.0, Cam[5].SegmentType := 1, Cam[6].Master := 61.0, Cam[6].Slave := 77.0, Cam[6].SegmentType := 1, Cam[7].Master := 90.0, Cam[7].SegmentType := 1, MasterPeriode := 90.0, SlavePeriode := 100.0, NbrOfCamPoints := 8, MasterScaling := 1.0, SlaveScaling := 1.0);
   Cam_Display_Verti : UDT_Axis_Cam_Profil := (Cam[0].Slave := 15.0, Cam[1].Master := 1.0, Cam[1].Slave := 15.0, Cam[2].Master := 6.0, Cam[2].Slave := 15.0, Cam[3].Master := 48.0, Cam[3].Slave := 15.0, Cam[3].SegmentType := 1, Cam[4].Master := 58.0, Cam[4].Slave := 25.0, Cam[5].Master := 63.0, Cam[5].Slave := 25.0, Cam[5].SegmentType := 1, Cam[6].Master := 81.0, Cam[6].Slave := 15.0, Cam[7].Master := 90.0, Cam[7].Slave := 15.0, Cam[7].SegmentType := 1, MasterPeriode := 90.0, SlavePeriode := 100.0, NbrOfCamPoints := 8, MasterScaling := 1.0, SlaveScaling := 1.0);
   CAM_Inter_Virtuel_Maitre : CAM[100] := ([1].Master := 90.0, [1].Slave := 90.0);
   CAM_Virtuel_Coupe_Fil : CAM[100] := ([1].Master := 90.0, [1].Slave := 360.0);
   CamGenerator_Coupe_Fil : AOI_CamGenerator_ST := (CycleTime := 12, L_NbCAMPoints := 3);
   CamGenerator_Horizontal : AOI_CamGenerator_ST := (CycleTime := 27, L_NbCAMPoints := 8);
   CamGenerator_Vertical : AOI_CamGenerator_ST := (CycleTime := 18, L_NbCAMPoints := 8);
   CF_Mode_Came_Activation : BOOL;
   CF_Mode_Came_Engagement : BOOL;
   CF_Mode_Top_Activation : BOOL := 1;
   CF_Mode_Top_Mouvement : BOOL;
   CO_Acquit_defaut : BOOL;
   CO_Activation : BOOL := 1;
   CO_Activation_Rouleaux : BOOL := 1;
   CO_Axe_Codeur_Four_Conv_Cons : REAL := 1000.0;
   CO_Axe_Codeur_Four_OK : BOOL := 1;
   CO_Axe_Codeur_Four_PosUnwind : DINT := 90000;
   CO_Axe_Coupe_Fil_Conv_Cons : REAL := 1000.0;
   CO_Axe_Coupe_Fil_OK : BOOL := 1;
   CO_Axe_Coupe_Fil_PosUnwind : DINT := 360000;
   CO_Axe_Horizontal_Droit_OK : BOOL := 1;
   CO_Axe_Horizontal_Gauche_OK : BOOL := 1;
   CO_Axe_Pompe_Doseuse_OK : BOOL := 1;
   CO_Axe_Reel_Desynchro : BOOL;
   CO_Axe_Reel_En_Synchro : BOOL := 1;
   CO_Axe_Rouleaux_Canneles_OK : BOOL := 1;
   CO_Axe_Vertical_Droit_OK : BOOL := 1;
   CO_Axe_Vertical_Gauche_OK : BOOL := 1;
   CO_Axe_Virtuel_Codeur_Conv_Cons : REAL := 1.0;
   CO_Axe_Virtuel_Codeur_PosUnwind : DINT := 90;
   CO_Axe_Virtuel_Maitre_Conv_Cons : REAL := 1.0;
   CO_Axe_Virtuel_Maitre_PosUnwind : DINT := 90;
   CO_BP_Coupe_Fil_Neg : BOOL;
   CO_BP_Coupe_Fil_Pos : BOOL;
   CO_BP_Horizontal_Droit_Neg : BOOL;
   CO_BP_Horizontal_Droit_Pos : BOOL;
   CO_BP_Horizontal_Gauche_Neg : BOOL;
   CO_BP_Horizontal_Gauche_Pos : BOOL;
   CO_BP_Pompe_Doseuse_Neg : BOOL;
   CO_BP_Pompe_Doseuse_Pos : BOOL;
   CO_BP_Rouleaux_Canneles_Neg : BOOL;
   CO_BP_Rouleaux_Canneles_Pos : BOOL;
   CO_BP_Vertical_Droit_Neg : BOOL;
   CO_BP_Vertical_Droit_Pos : BOOL;
   CO_BP_Vertical_Gauche_Neg : BOOL;
   CO_BP_Vertical_Gauche_Pos : BOOL;
   CO_Consigne_Pompe_Acc_Dec : REAL := 40.0;
   CO_Consigne_Pompe_Jerk : REAL := 100.0;
   CO_Consigne_Vitesse_Rouleaux : REAL := 0.41666666;
   CO_Control_Pompe_Vitesse : REAL := -0.16666667;
   CO_Defaut_ARU_Armoire : BOOL;
   CO_Defaut_ARU_Machine : BOOL;
   CO_Defaut_ARU_Pupitre : BOOL;
   CO_Defaut_CamGenerator_Coupe_Fil : BOOL;
   CO_Defaut_CamGenerator_Horizontal : BOOL;
   CO_Defaut_CamGenerator_Vertical : BOOL;
   CO_Defaut_Clef_Graissage : BOOL;
   CO_Defaut_CPT_Porte1 : BOOL;
   CO_Defaut_CPT_Porte2 : BOOL;
   CO_Defaut_CPT_Porte3 : BOOL;
   CO_Defaut_CPT_Porte4 : BOOL;
   CO_Defaut_Eth_Codeur_Four : BOOL;
   CO_Defaut_Eth_Var_Coupe_Fil : BOOL;
   CO_Defaut_Eth_Var_H_Droit : BOOL;
   CO_Defaut_Eth_Var_H_Gauche : BOOL;
   CO_Defaut_Eth_Var_Pompe_Doseuse : BOOL;
   CO_Defaut_Eth_Var_Rouleaux : BOOL;
   CO_Defaut_Eth_Var_V_Droit : BOOL;
   CO_Defaut_Eth_Var_V_Gauche : BOOL;
   CO_Defaut_FDC : BOOL;
   CO_Defaut_FDC_Amont_Horizontal_Droit : BOOL;
   CO_Defaut_FDC_Amont_Horizontal_Gauche : BOOL;
   CO_Defaut_FDC_Aval_Horizontal_Droit : BOOL;
   CO_Defaut_FDC_Aval_Horizontal_Gauche : BOOL;
   CO_Defaut_FDC_Bas_Vertical_Droit : BOOL;
   CO_Defaut_FDC_Bas_Vertical_Gauche : BOOL;
   CO_Defaut_FDC_Coupe_Fil_Droit : BOOL;
   CO_Defaut_FDC_Coupe_Fil_Gauche : BOOL;
   CO_Defaut_FDC_Haut_Vertical_Droit : BOOL;
   CO_Defaut_FDC_Haut_Vertical_Gauche : BOOL;
   CO_Defaut_Four : BOOL;
   CO_Defaut_Presence_Coupe_Fil : BOOL;
   CO_Defaut_Relais_Securite : BOOL;
   CO_Defauts_Secondaires : BOOL;
   CO_Degagement_En_Cours : BOOL;
   CO_Degagement_Possible : BOOL;
   CO_demande_darret : BOOL;
   CO_Demande_Init : BOOL;
   CO_en_Marche : BOOL := 1;
   CO_Engage_Axe_Coupe_Fil : Engage_Axe := (Activation := 1, Val_Vitesse := 100.0, Val_Acc := 1000.0, Val_Dec := 1000.0, Val_Jerk := 10000.0, Longeur_Cam := 3, Modulo_Maitre := 360.0, Mode_Rotatif := 1, Modulo_Esclave := 360, Axe_Degage := 1, Num_Cam_Vnul := 1);
   CO_Engage_Axe_H_Droit : Engage_Axe := (Activation := 1, Engagement := 1, Val_Vitesse := 50.0, Val_Acc := 500.0, Val_Dec := 500.0, Val_Jerk := 5000.0, Val_Degagement := 50.0, Longeur_Cam := 8, Modulo_Maitre := 90.0, Axe_Engage := 1, Num_Cam_Vnul := 1, Preposition_OK := 1);
   CO_Engage_Axe_H_Gauche : Engage_Axe := (Activation := 1, Engagement := 1, Val_Vitesse := 50.0, Val_Acc := 500.0, Val_Dec := 500.0, Val_Jerk := 5000.0, Val_Degagement := 50.0, Longeur_Cam := 8, Modulo_Maitre := 90.0, Axe_Engage := 1, Num_Cam_Vnul := 1, Changement_Came_Actif := 1, Preposition_OK := 1);
   CO_Engage_Axe_V_Droit : Engage_Axe := (Activation := 1, Engagement := 1, Engagement_Decalage := 1, Val_Vitesse := 50.0, Val_Acc := 500.0, Val_Dec := 500.0, Val_Jerk := 5000.0, Val_Engagement := -14.0, Val_Degagement := 35.0, Val_Decalage := -14.0, Longeur_Cam := 8, Modulo_Maitre := 90.0, Axe_Engage := 1, Preposition_OK := 1);
   CO_Engage_Axe_V_Gauche : Engage_Axe := (Activation := 1, Engagement := 1, Engagement_Decalage := 1, Val_Vitesse := 50.0, Val_Acc := 500.0, Val_Dec := 500.0, Val_Jerk := 5000.0, Val_Engagement := -14.0, Val_Degagement := 35.0, Val_Decalage := -14.0, Longeur_Cam := 8, Modulo_Maitre := 90.0, Axe_Engage := 1, Num_Cam_Vnul := 1, Preposition_OK := 1);
   CO_Engage_Maitre : Engage_Axe_Virtuel := (Activation := 1, Engagement := 1, Val_Vitesse := 3600.0, Val_Acc := 100000.0, Val_Dec := 100000.0, Val_Jerk := 360000.0, Longeur_Cam := 2, Modulo_Maitre := 90.0, Modulo_Esclave := 90, Axe_Engage := 1);
   CO_Engage_Virtuel_Coupe_Fil : Engage_Axe_Virtuel := (Val_Vitesse := 3600.0, Val_Acc := 100000.0, Val_Dec := 100000.0, Val_Jerk := 360000.0, Longeur_Cam := 2, Modulo_Maitre := 90.0, Modulo_Esclave := 360, Axe_Degage := 1);
   CO_Engagement : BOOL := 1;
   CO_Engagement_Coupe_Fil : BOOL;
   CO_Engagement_Maitre : BOOL := 1;
   CO_Ethernet_Code_Def_Codeur_Four : DINT;
   CO_Ethernet_Code_Def_Coupe_Fil : DINT;
   CO_Ethernet_Code_Def_H_Droit : DINT;
   CO_Ethernet_Code_Def_H_Gauche : DINT;
   CO_Ethernet_Code_Def_Pompe_Doseuse : DINT;
   CO_Ethernet_Code_Def_Rouleaux : DINT;
   CO_Ethernet_Code_Def_V_Droit : DINT;
   CO_Ethernet_Code_Def_V_Gauche : DINT;
   CO_Flip_100ms : TIMER := (PRE := 50, ACC := 40, EN := 1, TT := 1);
   CO_Flip_500ms : TIMER := (PRE := 500, ACC := 500, EN := 1, DN := 1);
   CO_Flop_100ms : TIMER := (PRE := 50);
   CO_Flop_500ms : TIMER := (PRE := 500, ACC := 420, EN := 1, TT := 1);
   CO_Front_Activation : BOOL := 1;
   CO_Front_Demande_Init : BOOL;
   CO_Front_Raz_Init : BOOL;
   CO_Front_Reset_Init_OK : BOOL;
   CO_Init_Coupe_Fil : BOOL;
   CO_Init_Horizontal_Droit : BOOL;
   CO_Init_Horizontal_Gauche : BOOL;
   CO_Init_Ok : BOOL := 1;
   CO_Init_Pompe_Doseuse : BOOL;
   CO_Init_Rouleaux_Canneles : BOOL;
   CO_Init_Vertical_Droit : BOOL;
   CO_Init_Vertical_Gauche : BOOL;
   CO_Machine_sans_defaut : BOOL := 1;
   CO_MAH_Virtuel_Coupe_Fil : MOTION_INSTRUCTION := (FLAGS := 704643072, DN := 1, PC := 1, STATE := 17);
   CO_Marche : BOOL := 1;
   CO_Messages_En : STRING[380] := ([0] := 'No Axis Error Pending', [3] := 'Err3: Execution Collision', [4] := 'Err4: Open the servo loop before you execute this instruction', [5] := 'Err5: Close the servo loop before you execute this instruction', [7] := 'Err7: Shutdown State Error', [8] := 'Err8: Wrong Axis Type', [9] := 'Err9: Overtravel condition.', [10] := 'Err10: Master Axis Conflict', [11] := 'Err11: Axis Not Configured', [12] := 'Err12: Servo Message Failure', [13] := 'Err13: Parameter Out Of Range', [14] := 'Err14: Tune Process Error', [15] := 'Err15: Test Process Error', [16] := 'Err16: Home In Process Error', [17] := 'Err17: Axis Mode Not Rotary', [18] := 'Err18: Axis Type Unused', [19] := 'Err19: Axis Group Not Synchronized', [20] := 'Err20: Axis In Faulted State', [21] := 'Err21: Group in Faulted State', [22] := 'Err22: Axis in Motion', [23] := 'Err23: Illegal Dynamic Change', [24] := 'Err24: Illegal Controller Mode Operation', [25] := 'Err25: Illegal Instruction', [26] := 'Err26: Illegal Cam Length', [27] := 'Err27: Illegal Cam Profile Length', [28] := 'Err28: Illegal Cam Type', [29] := 'Err29: Illegal Cam Order', [30] := 'Err30: Cam Profile Being Calculated', [31] := 'Err31: Cam Profile Being Used', [32] := 'Err32: Cam Profile Not Calculated', [33] := 'Err33: Position Cam Not Enabled', [34] := 'Err34: Registration in Progress', [35] := 'Err35: Illegal Execution Target', [36] := 'Err36: Illegal Output Cam', [37] := 'Err37: Illegal Output Compensation', [38] := 'Err38: Illegal Axis Data Type', [39] := 'Err39: Process Conflict', [40] := 'Err40: Drive Locally Disabled', [41] := 'Err41: Illegal Homing Configuration', [42] := 'Err42: ShutDown Status TimeOut', [43] := 'Err43: Coordinate System Queue Full', [44] := 'Err44: Circular Collinearity Error', [45] := 'Err45: Circular Start End ', [46] := 'Err46: Circular R1 R2 Mismatch Error', [47] := 'Err47: Circular Infinite Solution Error', [48] := 'Err48: Circular No Solutions Error', [49] := '49: Circular Small R Error', [50] := 'Err50: Coordinate System Not in Group', [51] := 'Err51: Invalid Actual Tolerance', [52] := 'Err52: Coordination Motion In Process Error', [53] := 'Err53: Axis Is Inhibited', [54] := 'Err54: Deceleration Is Set To ZERO', [61] := 'Err61: Connection Conflict', [62] := 'Err62: Transform In Progress', [63] := 'Err63: Axis In Transform Motion', [64] := 'Err64: Ancillary Not Supported', [65] := 'Err65: Axis Position Overflow', [66] := 'Err66: Robot Movmnt not Allowed', [67] := 'Err67: Invalid Transform Position', [68] := 'Err68: Transform At Origin',
        [69] := 'Err69: Max Joint Velocity Exceeded', [70] := 'Err70: Axes In Transform Must Be Linear', [71] := 'Err71: Transform Is Canceling', [72] := 'Err72: Max Joint Angle Exceeded', [73] := 'Err73: Coord System Chaining Error', [74] := 'Err74: Invalid Orientation Angle', [75] := 'Err75: Instruction Not Supported', [76] := 'Err76: Deceleration Jerk Is Set To ZERO', [77] := 'Err77: Transform Direction Not Supported', [100] := 'Pos Soft Overtravel Fault', [101] := 'Neg Soft Overtravel Fault', [102] := 'Pos Hard Overtravel Fault', [103] := 'Neg Hard Overtravel Fault', [104] := 'Motor FeedBack Fault', [105] := 'Motor FeedBack Noise', [106] := 'Aux FeedBack Fault', [107] := 'Aux FeedBack Noise', [108] := 'Reserved', [109] := 'Drive Enable Input Fault', [110] := 'Common DC Bus Fault', [111] := 'DC Bus Precharge Overload Fault', [112] := 'Reserved', [113] := 'Ground ShortCut Fault', [114] := 'Drive Hard Fault', [115] := 'OverSpeed Fault', [116] := 'Overload Fault I2T', [117] := 'Drive Over Temperature', [118] := 'Motor Over Temperature', [119] := 'Drive Cooling Fault', [120] := 'Drive Cooling Voltage Fault', [121] := 'FeedBack Fault', [122] := 'Communication Fault', [123] := 'Drive Over Current Fault', [124] := 'Drive Over Voltage Fault', [125] := 'Drive Under Voltage Fault', [126] := 'Phase Power Supply Fault or Loss', [127] := 'Following Error Fault', [128] := 'SERCOS Fault', [129] := 'Overtravel Fault', [130] := 'Reserved', [131] := 'Manufacturer Specific Fault', [134] := 'Motor Commutation Fault', [135] := 'Motor Overspeed FL Fault', [136] := 'Motor Overspeed UL Fault', [137] := 'Motor Overtemperature FL Fault', [138] := 'Motor Overtemperature UL Fault', [139] := 'Motor Thermal Overload FL Fault', [140] := 'Motor Thermal Overload UL Fault', [141] := 'Inverter Overcurrent Fault', [142] := 'Inverter Overtemperature FL Fault', [143] := 'Inverter Overtemperature UL Fault', [144] := 'Inverter Thermal Overload FL Fault', [145] := 'Inverter Thermal Overload UL Fault', [146] := 'Converter Ground Current FL Fault', [147] := 'Converter Ground Current UL Fault', [148] := 'Converter Overtemperature FL Fault', [149] := 'Converter Overtemperature UL Fault', [150] := 'Converter Thermal Overload FL Fault', [151] := 'Converter Thermal Overload UL Fault', [152] := 'Converter AC Power Loss Fault',
        [153] := 'Converter AC Single Phase Loss Fault', [154] := 'Converter AC Phase Short Fault', [155] := 'Converter Pre Charge Fault', [156] := 'Bus Regulator Overtemperature FL Fault', [157] := 'Bus Regulator Overtemperature UL Fault', [158] := 'Bus Regulator Thermal Overload FL Fault', [159] := 'Bus Regulator Thermal Overload UL Fault', [160] := 'Bus Undervoltage FL Fault', [161] := 'Bus Undervoltage UL Fault', [162] := 'Bus Overvoltage FL Fault', [163] := 'Bus Overvoltage UL Fault', [164] := 'Bus Power Loss Fault', [165] := 'Bus Power Blown Fuse', [166] := 'Feedback Signal Noise FL Fault', [167] := 'Feedback Signal Noise UL Fault', [168] := 'Feedback Signal Loss FL Fault', [169] := 'Feedback Signal Loss UL Fault', [170] := 'Feedback Data Loss FL Fault', [171] := 'Feedback Data Loss UL Fault', [172] := 'Feedback Device Fault', [173] := 'Hardware Overtravel Positive Fault', [174] := 'Hardware Overtravel Negative Fault', [175] := 'Excessive Position Error Fault', [176] := 'Excessive Velocity Error Fault', [177] := 'Overtorque Limit Fault', [178] := 'Undertorque Limit Fault', [179] := 'Illegal Control Mode Fault', [180] := 'Enable Input Deactivated Fault', [181] := 'Controller Initiated Fault', [182] := 'External Input Fault', [183] := 'Commutation Startup Failure', [184] := 'Motor Voltage Mismatch', [185] := 'Feedback Filter Noise', [186] := 'Feedback Battery Loss', [187] := 'Feedback Batter Low', [188] := 'Feedback Incremental Count Error', [189] := 'Control Module Overtemperature FL', [190] := 'Control Module Overtemperature UL', [191] := 'Converter Pre-charge Overload FL', [192] := 'Converter Pre-charge Overload UL', [193] := 'Excessive Current Feedback Fault', [194] := 'Regenerative Power Supply Fault', [195] := 'PWM Frequency Reduced Fault', [196] := 'Current Limit Reduced Fault', [197] := 'Torque Prove Fault', [198] := 'Decel Override Fault', [199] := 'Preventative Maintenance Fault', [200] := 'Axis Not Enable', [201] := 'Axis Enabled, No OpMode', [202] := 'Wait For Start', [203] := 'Homing Processing', [204] := 'Homing Done', [205] := 'Wait For JogFw Or JobBw', [206] := 'Jogging Forward', [207] := 'Jogging Backward', [208] := 'Moving Endless', [209] := 'Moving To Stop Position', [210] := 'Moving To Target', [211] := 'Procedure Aborded', [212] := 'Position Reached',
        [213] := 'Procedure Stopped', [214] := 'Remove Start Command', [215] := 'Wait For RecoverStart', [216] := 'Remove RecoverStart', [217] := 'Moving To Synchronisation Position', [218] := 'Synchronised To The Master By CamProfil', [220] := 'StopMode 1 Is Active', [221] := 'StopMode 2 Is Active', [222] := 'StopMode 3 is Active', [223] := 'StopMode 4 is Active', [224] := 'Safe Torque Off Active', [225] := 'HWLimitPos Active', [226] := 'HWLimitNeg Active', [230] := 'Synchronised, Ready For NewCam', [231] := 'Changing CamProfil', [240] := 'Motor Test Fault', [241] := 'Hardware Configuration Fault', [242] := 'Firmware Change Fault', [243] := 'DC Common Bus Fault', [244] := 'Runtime Error Fault', [245] := 'Backplane Communication Error Fault', [246] := 'Safety Module Communication Error Fault', [247] := 'Product Specific Fault', [250] := 'Module Fault : Control Sync Fault', [251] := 'Module Fault : Module Sync Fault', [252] := 'Module Fault : Timer Event Fault', [253] := 'Module Fault : Module Hard Fault', [254] := 'Module Fault : Module Connection Fault', [255] := 'Module Fault : Connection Format Fault', [256] := 'Module Fault : Local Mode Fault', [257] := 'Module Fault : CPU Watchdog Fault', [258] := 'Module Fault : Clock Jitter Fault', [259] := 'Module Fault : Cyclic Read Fault', [260] := 'Module Fault : Cyclic Write Fault', [261] := 'Module Fault : Clock Skew Fault', [262] := 'Module Fault : Control Connection Fault', [263] := 'Module Fault : Control Clock Sync Fault', [264] := 'Module Fault : Module Clock Sync Fault', [265] := 'Module Fault : Logic Watchdog Fault', [266] := 'Module Fault : Duplicate Address Fault', [270] := 'Config Fault : Connection failure', [271] := 'Config Fault : Resource unavailable', [272] := 'Config Fault : Invalid value in object specific data param of a service request', [273] := 'Config Fault : IOI segment error', [274] := 'Config Fault : IOI destination unknown', [275] := 'Config Fault : Partial transfer', [276] := 'Config Fault : Connection lost', [277] := 'Config Fault : Unimplemented service', [278] := 'Config Fault : Invalid attribute value', [279] := 'Config Fault : Attribute list error', [280] := 'Config Fault : Already in requested mode/state', [281] := 'Config Fault : Object can not perform service in its current mode/state', [282] := 'Config Fault : Object already exists', [283] := 'Config Fault : Attribute value not settable', [284] := 'Config Fault : Access permission does not allow service', [285] := 'Config Fault : Devices mode/state does not allow object to perform service', [286] := 'Config Fault : Reply data too large', [287] := 'Config Fault : Fragmentation of a primitive value', [288] := 'Config Fault : Not enough data', [289] := 'Config Fault : Undefined attribute',
        [290] := 'Config Fault : Too much data', [291] := 'Config Fault : Object does not exist', [292] := 'Config Fault : Service fragmentation sequence not currently in progress', [293] := 'Config Fault : No stored attribute data', [294] := 'Config Fault : Store operation failure', [295] := 'Config Fault : Bridging failure, request packet too large for network', [296] := 'Config Fault : Bridging failure, response packet too large for network', [297] := 'Config Fault : Missing attribute list entry data', [298] := 'Config Fault : Invalid attribute value list', [299] := 'Config Fault : Embedded service error', [300] := 'Config Fault : Connection Related Failure', [301] := 'Config Fault : Invalid Parameter', [302] := 'Config Fault : Writeonce value or medium already written', [303] := 'Config Fault : Invalid Reply Received', [304] := 'Config Fault : CST not coordinated', [305] := 'Config Fault : Connection Scheduling Error', [306] := 'Config Fault : Key Failure in IOI', [307] := 'Config Fault : IOI Size Invalid', [308] := 'Config Fault : Unexpected attribute in list', [309] := 'Config Fault : DNet Invalid Member ID', [310] := 'Config Fault : DNet Member not settable', [311] := 'Group Fault', [312] := 'Guard Internal Fault', [313] := 'Guard Configuration Fault', [314] := 'Guard Gate Drive Fault', [315] := 'Guard Reset Fault', [316] := 'Guard Feedback 1 Fault', [317] := 'Guard Feedback 2 Fault', [318] := 'Guard Feedback Speed Compare Fault', [319] := 'Guard Feedback Position Compare Fault', [320] := 'Guard Stop Input Fault', [321] := 'Guard Stop Output Fault', [322] := 'Guard Stop Decel Fault', [323] := 'Guard Stop Standstill Fault', [324] := 'Guard Stop Motion Fault', [325] := 'Guard Limited Speed Input Fault', [326] := 'Guard Limited Speed Output Fault', [327] := 'Guard Limited Speed Monitor Fault', [328] := 'Guard Max Speed Monitor Fault', [329] := 'Guard Max Accel Monitor Fault', [330] := 'Guard Direction Monitor Fault', [331] := 'Guard Door Monitor Input Fault', [332] := 'Guard Door Monitor Fault', [333] := 'Guard Door Control Output Fault', [334] := 'Guard Lock Monitor Input Fault', [335] := 'Guard Lock Monitor Fault', [336] := 'Guard Enabling Switch Monitor Input Fault', [337] := 'Guard Enabling Switch Monitor Fault', [338] := 'Guard Feedback 1 Voltage Monitor Fault', [339] := 'Guard Feedback 2 Voltage Monitor Fault', [340] := 'Init Fault : Boot Block Checksum Fault', [341] := 'Init Fault : Main Block Checksum Fault', [342] := 'Init Fault : Nonvolatile Memory Checksum Fault', [343] := 'Init Fault : Commutation Not Configured', [344] := 'Init Fault : Feedback Data Corruption', [345] := 'Init Fault : Feedback Data Range', [346] := 'Init Fault : Feedback Communication Startup', [347] := 'Init Fault : Feedback Absolute Overspeed', [348] := 'Init Fault : Feedback Absolute Power Off Travel', [349] := 'Init Fault : Feedback Absolute Startup Speed',
        [350] := 'Init Fault : Commutation Offset Uninitialized', [351] := 'Init Fault : Invalid FPGA Image', [352] := 'Init Fault : Invalid Board Support Package', [353] := 'Init Fault : Invalid Safety Firmware', [354] := 'Init Fault : Power Board', [355] := 'Init Fault : Illegal Option Card', [356] := 'Init Fault : Option Storage Checksum', [357] := 'Init Fault : Module Voltage Mismatch', [358] := 'Init Fault : Unknown Module', [359] := 'Init Fault : Factory Configuration Error', [360] := 'Init Fault : Illegal Address', [361] := 'Init Fault : Series Mismatch', [362] := 'Init Fault : Open Slot', [363] := 'APR Fault');
   CO_Pilotage_Coupe_Fil : Pilotage_Relatif_Virtuel := (MVT_Activation := 1, MVT_Val_Position := 360.0, MVT_Val_Vitesse := 200.0, MVT_Val_Acc := 1000.0, MVT_Val_Dec := 1000.0, MVT_Val_Jerk := 50.0, MVT_En_Pos := 1, MVT_Mode_Positionnement := 1, MVT_Tolerance_Arret := 10.0, MVT_Axe_Modulo := 1, MVT_Val_Modulo := 360);
   CO_Pilotage_Pompe_Doseuse : Pilotage_Relatif := (MVT_Val_Vitesse := 1.0, MVT_En_Pos := 1, MVT_Mode_Positionnement := 1, MVT_Tolerance_Arret := 10.0, MVT_Axe_Modulo := 1, MVT_Val_Modulo := 360);
   CO_Raz_Axe : BOOL;
   CO_Synchro_Axe_En_Cours : BOOL;
   CO_Temp_Activation : TIMER := (PRE := 1500, ACC := 1500, EN := 1, DN := 1);
   CO_Temp_Desynchro : TIMER := (PRE := 500);
   CO_Temp_Pret : TIMER := (PRE := 1500, ACC := 1500, EN := 1, DN := 1);
   CO_Temp_Vitesse_Four : REAL := 2791.1553;
   CO_Tempo_Demande_Init : TIMER := (PRE := 2500);
   CO_Tempo_Engagement : TIMER := (PRE := 500, ACC := 500, EN := 1, DN := 1);
   CO_Tempo_Valid_Recette : TIMER := (PRE := 5000, ACC := 5000);
   CO_Temps_de_demarrage : TIMER;
   CO_TOF_Top_Decoreuse : TIMER := (PRE := 500, ACC := 500);
   CO_TOF_Top_Doseuse : TIMER := (PRE := 500, ACC := 500);
   CO_TON_Activation : TIMER := (PRE := 500, ACC := 500, EN := 1, DN := 1);
   CO_Top_Debut_Cycle_Decoreuse : BOOL;
   CO_Top_Debut_Dosage : BOOL;
   CO_Top_Degagement : BOOL;
   CO_Top_Depart_Coupe_Fil : BOOL;
   CO_Top_Depart_Pompe : BOOL;
   CO_Top_Depart_Pompe_Avance : BOOL;
   CO_Top_Depart_Pompe_Inter1 : BOOL;
   CO_Top_Depart_Pompe_Inter2 : BOOL;
   CO_Top_Depart_Pompe_Inter3 : BOOL;
   CO_Top_Depart_Pompe_Inter4 : BOOL;
   CO_Top_Depart_Pompe_Inter5 : BOOL;
   CO_Top_Depart_Pompe_Inter6 : BOOL;
   CO_Top_Depart_Pompe_Inter7 : BOOL;
   CO_Top_Depart_Pompe_Inter8 : BOOL;
   CO_Top_Depart_Pompe_Recul : BOOL := 1;
   CO_Top_Depart_Rouleaux : BOOL;
   CO_Top_Once_Axe_Virtuel : BOOL;
   CO_Top_Once_Decoreuse : BOOL;
   CO_Top_Once_Doseuse : BOOL;
   CO_Top_Recalage : BOOL;
   CO_Validation_Recette : BOOL;
   Com_Comas_Conv : DINT[10] := ([0] := 1, [1] := 4604, [2] := 2783);
   Com_Comas_Conv_ASUPP : DINT := 1;
   Com_Comas_Gen_Conv : DINT[10] := ([0] := 40, [2] := 1000001984, [4] := 3);
   Com_Comas_Sortie_F : UDT_COM_Comas_Vers_SortieF; {produced}
   Consigne_Acc_Decc_Manu_Degre : DINT := 3600;
   Consigne_Vitesse_Manu_Degre_Seconde : REAL := 60.0;
   Consigne_Vitesse_Manu_Tour_Seconde : REAL := 0.16666667;
   Correction_Vitesse_Virtuel : REAL;
   Cpt_Delta_Codeur : REAL := 4198.582;
   Cpt_Det_Produit : REAL;
   Cpt_Det_Produit2 : REAL := 50000.074;
   Cpt_Fin_Det_Produit : REAL := 50000.16;
   Cpt_Fin_Det_Produit2 : REAL;
   Cpt_Mini_Entre_Produit : REAL := 50000.016;
   Cpt_Mini_Entre_Produit2 : REAL := 50000.074;
   Delta_Avance_Tapis_Four : REAL := 0.23900032;
   Det_Produit : BOOL;
   Det_Produit2 : BOOL;
   DFE : BOOL;
   Distance_CPT_Presence_Produit : DINT := 520;
   Distance_Decoreuse : DINT;
   Distance_Doseuse : DINT;
   ENT_Badge_Code_A : ALIAS FOR Local:1:I.Pt11.Data;
   ENT_Badge_Code_B : ALIAS FOR Local:1:I.Pt12.Data;
   ENT_Badge_Code_C : ALIAS FOR Local:1:I.Pt13.Data;
   ENT_Badge_Code_D : ALIAS FOR Local:1:I.Pt14.Data;
   ENT_Badge_STR : ALIAS FOR Local:1:I.Pt15.Data;
   ENT_CO_ARU_Armoire : ALIAS FOR Local:1:I.Pt03.Data;
   ENT_CO_ARU_Machine : ALIAS FOR Local:1:I.Pt05.Data;
   ENT_CO_ARU_Pupitre : ALIAS FOR Local:1:I.Pt04.Data;
   ENT_CO_BP_Arret : ALIAS FOR Local:1:I.Pt01.Data;
   ENT_CO_BP_Marche : ALIAS FOR Local:1:I.Pt00.Data;
   ENT_CO_BP_Rearmement : ALIAS FOR Local:1:I.Pt02.Data;
   ENT_CO_Clef_Graissage : ALIAS FOR Local:2:I.Pt02.Data;
   ENT_CO_CPT_Porte1 : ALIAS FOR Local:1:I.Pt06.Data;
   ENT_CO_CPT_Porte2 : ALIAS FOR Local:1:I.Pt07.Data;
   ENT_CO_CPT_Porte3 : ALIAS FOR Local:1:I.Pt08.Data;
   ENT_CO_CPT_Porte4 : ALIAS FOR Local:1:I.Pt09.Data;
   ENT_CO_CPT_Presence_Produit : ALIAS FOR Local:2:I.Pt07.Data;
   ENT_CO_FDC_Amont_Horizontal_Droit : ALIAS FOR Local:2:I.Pt15.Data;
   ENT_CO_FDC_Amont_Horizontal_Gauche : ALIAS FOR Local:2:I.Pt13.Data;
   ENT_CO_FDC_Aval_Horizontal_Droit : ALIAS FOR Local:2:I.Pt14.Data;
   ENT_CO_FDC_Aval_Horizontal_Gauche : ALIAS FOR Local:2:I.Pt12.Data;
   ENT_CO_FDC_Bas_Vertical_Droit : ALIAS FOR Local:2:I.Pt10.Data;
   ENT_CO_FDC_Bas_Vertical_Gauche : ALIAS FOR Local:2:I.Pt08.Data;
   ENT_CO_FDC_Coupe_Fil_Droit : BOOL;
   ENT_CO_FDC_Coupe_Fil_Gauche : BOOL;
   ENT_CO_FDC_Haut_Vertical_Droit : ALIAS FOR Local:2:I.Pt11.Data;
   ENT_CO_FDC_Haut_Vertical_Gauche : ALIAS FOR Local:2:I.Pt09.Data;
   ENT_CO_Presence_Coupe_Fil : ALIAS FOR Local:2:I.Pt00.Data;
   ENT_CO_Relais_Securite : ALIAS FOR Local:1:I.Pt10.Data;
   ENT_CPT_Synchronisme : ALIAS FOR Local:2:I.Pt06.Data;
   ENT_CPT_Synchronisme2 : ALIAS FOR Local:2:I.Pt05.Data;
   ENT_Four_OK : ALIAS FOR Local:2:I.Pt01.Data;
   ENT_Reisdorf_en_Marche : ALIAS FOR Local:2:I.Pt03.Data;
   Fin_Rouleau : REAL := 41.0;
   Flip_Display : TIMER := (PRE := 500, ACC := 500, EN := 1, DN := 1);
   Flop_Display : TIMER := (PRE := 500, ACC := 425, EN := 1, TT := 1);
   Front_Badge : BOOL := 1;
   Front_Cpt_Det_PRoduit : FBD_ONESHOT;
   Front_Cpt_Det_PRoduit2 : FBD_ONESHOT := (InputBit := 1);
   Front_Det_produit : FBD_ONESHOT;
   Front_Det_produit2 : FBD_ONESHOT := (InputBit := 1);
   Front_Det_produit_2 : BOOL;
   Front_Det_Produit_Filtre : FBD_ONESHOT;
   Front_Det_Produit_Filtre2 : FBD_ONESHOT;
   Front_Det_produit_Moyennage : BOOL;
   Front_Det_produit_Moyennage2 : BOOL;
   Front_Det_produit_Resynchro : BOOL := 1;
   Front_Det_produit_Resynchro2 : BOOL;
   Front_Moyennage_Cadencement : FBD_ONESHOT;
   Front_Resynchro_temp : BOOL;
   Front_Top_Recalage : BOOL;
   Front_Valid_Recette : BOOL;
   g_Modulo_Codeur_Four : DINT := 90;
   g_Unwind_Axe_Codeur_Four : DINT := 90000;
   index_moyennage : DINT := 151;
   index_recette : DINT := 50;
   Index_Tableau_Tapis : DINT;
   Init_Coupe_Fil : Init_Axe_CIP := (Vitesse := 20.0, Acc := 200.0, Dec := 200.0, Jerk := 2000.0, Init_OK := 1);
   Init_Horizontal_Droit : Init_Axe_CIP := (Vitesse := 2.0, Acc := 20.0, Dec := 20.0, Jerk := 200.0, Init_OK := 1);
   Init_Horizontal_Gauche : Init_Axe_CIP := (Vitesse := 2.0, Acc := 20.0, Dec := 20.0, Jerk := 200.0, Init_OK := 1);
   Init_Pompe_Doseuse : Init_Axe_CIP := (Vitesse := 0.1, Acc := 50.0, Dec := 50.0, Jerk := 500.0, Init_OK := 1);
   Init_Rouleaux_Canneles : Init_Axe_CIP := (Vitesse := 20.0, Acc := 50.0, Dec := 50.0, Jerk := 500.0);
   Init_Vertical_Droit : Init_Axe_CIP := (Vitesse := 2.0, Acc := 20.0, Dec := 20.0, Jerk := 200.0, Init_OK := 1);
   Init_Vertical_Gauche : Init_Axe_CIP := (Vitesse := 2.0, Acc := 20.0, Dec := 20.0, Jerk := 200.0, Init_OK := 1);
   L_Ms_Index_Codeur_Four : DINT;
   L_Ms_Index_Coupe_Fil : DINT;
   L_Ms_Index_H_Droit : DINT;
   L_Ms_Index_H_Gauche : DINT;
   L_Ms_Index_Pompe_Doseuse : DINT;
   L_Ms_Index_Rouleaux : DINT;
   L_Ms_Index_V_Droit : DINT;
   L_Ms_Index_V_Gauche : DINT;
   Lecteur_Badge_Code_A : BOOL;
   Lecteur_Badge_Code_B : BOOL;
   Lecteur_Badge_Code_C : BOOL;
   Lecteur_Badge_Code_D : BOOL;
   Longueur_Maxi_Tapis_Four : REAL := 10000.0;
   MAM_Correction_Cod_Virtuel : MOTION_INSTRUCTION := (FLAGS := 268435456, ER := 1, ERR := 11, EXERR := 1);
   MAM_Correction_Cod_Virtuel_test : MOTION_INSTRUCTION := (FLAGS := 536870912, DN := 1);
   MAM_Correction_Cod_Virtuel_test2 : MOTION_INSTRUCTION := (FLAGS := 536870912, DN := 1);
   MAM_Resyncho_Codeur : MOTION_INSTRUCTION := (FLAGS := 33554432);
   MAM_Resynchro_Accel_Correction : REAL := 200.0;
   MAM_Resynchro_Vitesse_Correction : REAL := 20.0;
   Memo_Recalage_Detection_PRoduit_1 : BOOL;
   Memo_Recalage_Detection_PRoduit_2 : BOOL;
   Message_Axe_Codeur_Four : Message_Axe;
   Message_Axe_Coupe_Fil : Message_Axe;
   Message_Axe_H_Droit : Message_Axe;
   Message_Axe_H_Gauche : Message_Axe;
   Message_Axe_Pompe_Doseuse : Message_Axe;
   Message_Axe_Rouleaux : Message_Axe;
   Message_Axe_V_Droit : Message_Axe;
   Message_Axe_V_Gauche : Message_Axe;
   Message_Defaut_Codeur_Four : STRING := 'No Axis Error Pending';
   Message_Defaut_Coupe_Fil : STRING := 'No Axis Error Pending';
   Message_Defaut_H_Droit : STRING := 'No Axis Error Pending';
   Message_Defaut_H_Gauche : STRING := 'No Axis Error Pending';
   Message_Defaut_Pompe_Doseuse : STRING := 'No Axis Error Pending';
   Message_Defaut_Rouleaux : STRING := 'No Axis Error Pending';
   Message_Defaut_V_Droit : STRING := 'No Axis Error Pending';
   Message_Defaut_V_Gauche : STRING := 'No Axis Error Pending';
   MSG_General_Convoyage : MESSAGE;
        MessageParameters(ServiceCode := 16#004c, LocalElement := Com_Comas_Gen_Conv[0], ...)
   MSG_Vitesse_Four_L4 : MESSAGE;
        MessageParameters(ServiceCode := 16#004c, LocalElement := Vitesse_Four4_Real, ...)
   Output_Cams_Coupe_Fil : Output_Cams := (In_ServoPos := 30.0, Set_Period := 90.0, Set_OnPos := 11.0, Set_OffPos := 21.0);
   Output_Cams_Decoreuse : Output_Cams := (Cmd_Enable_AOI := 1, In_ServoPos := 71.0, In_ServoVel := 200.0, Set_Period := 90.0);
   Output_Cams_Degagement : Output_Cams := (Cmd_Enable_AOI := 1, In_ServoPos := 24.0, In_ServoVel := 200.0, Set_Period := 90.0, Set_OffPos := 10.0);
   Output_Cams_Dosage : Output_Cams := (Cmd_Enable_AOI := 1, In_ServoPos := 62.0, Set_Period := 90.0);
   Output_Cams_Pompe_Avance : Output_Cams := (Cmd_Enable_AOI := 1, In_ServoPos := 80.0, Set_Period := 90.0, Set_OnPos := -19.0, Set_OffPos := 31.0, Out_Cam := 1);
   Output_Cams_Pompe_Inter1 : Output_Cams := (In_ServoPos := 38.0, Set_Period := 100.0);
   Output_Cams_Pompe_Inter2 : Output_Cams := (In_ServoPos := 38.0, Set_Period := 100.0);
   Output_Cams_Pompe_Inter3 : Output_Cams := (In_ServoPos := 38.0, Set_Period := 100.0);
   Output_Cams_Pompe_Inter4 : Output_Cams := (In_ServoPos := 38.0, Set_Period := 100.0);
   Output_Cams_Pompe_Inter5 : Output_Cams := (In_ServoPos := 38.0, Set_Period := 100.0);
   Output_Cams_Pompe_Inter6 : Output_Cams := (In_ServoPos := 38.0, Set_Period := 100.0);
   Output_Cams_Pompe_Inter7 : Output_Cams := (In_ServoPos := 38.0, Set_Period := 100.0);
   Output_Cams_Pompe_Inter8 : Output_Cams := (In_ServoPos := 38.0, Set_Period := 100.0);
   Output_Cams_Pompe_Recul : Output_Cams := (Cmd_Enable_AOI := 1, In_ServoPos := 43.0, Set_Period := 90.0, Set_OnPos := 43.0, Set_OffPos := 63.0);
   Output_Cams_Recalage : Output_Cams := (Cmd_Enable_AOI := 1, In_ServoPos := 16.0, In_ServoVel := 200.0, Set_Period := 90.0, Set_OnPos := -19.0, Set_OffPos := 41.0, Out_Cam := 1);
   Output_Cams_Rouleaux : Output_Cams := (Cmd_Enable_AOI := 1, In_ServoPos := 8.0, Set_Period := 90.0, Set_OnPos := -19.0, Set_OffPos := 31.0, Out_Cam := 1);
   PCAM_Coupe_Fil : UDT_CamGeneration := (In.Cam[0].SegmentType := 1, In.Cam[1].Master := 180.0, In.Cam[1].Slave := 90.0, In.Cam[2].Master := 360.0, In.Cam[2].Slave := 360.0, In.Cam[2].SegmentType := 1, Out.Cam[0].SegmentType := 1, Out.Cam[1].Master := 180.0, Out.Cam[1].Slave := 90.0, Out.Cam[2].Master := 360.0, Out.Cam[2].Slave := 360.0, Out.Cam[2].SegmentType := 1, Out.NbrOfCamPoints := 3, Out.CamProfil[0].Status := 2, Out.CamProfil[1].Status := 2, Out.CamProfil[2].Status := 2);
   PCAM_Horizontal : UDT_CamGeneration := (In.Cam[1].Master := 1.0, In.Cam[1].SegmentType := 1, In.Cam[2].Master := 6.0, In.Cam[2].Slave := 5.0, In.Cam[3].Master := 36.0, In.Cam[3].Slave := 77.0, In.Cam[3].SegmentType := 1, In.Cam[4].Master := 46.0, In.Cam[4].Slave := 87.0, In.Cam[5].Master := 51.0, In.Cam[5].Slave := 87.0, In.Cam[5].SegmentType := 1, In.Cam[6].Master := 61.0, In.Cam[6].Slave := 77.0, In.Cam[6].SegmentType := 1, In.Cam[7].Master := 90.0, Out.Cam[1].Master := 1.0, Out.Cam[1].SegmentType := 1, Out.Cam[2].Master := 6.0, Out.Cam[2].Slave := 5.0, Out.Cam[3].Master := 36.0, Out.Cam[3].Slave := 77.0, Out.Cam[3].SegmentType := 1, Out.Cam[4].Master := 46.0, Out.Cam[4].Slave := 87.0, Out.Cam[5].Master := 51.0, Out.Cam[5].Slave := 87.0, Out.Cam[5].SegmentType := 1, Out.Cam[6].Master := 61.0, Out.Cam[6].Slave := 77.0, Out.Cam[6].SegmentType := 1, Out.Cam[7].Master := 90.0, Out.Cam[7].SegmentType := 1, Out.NbrOfCamPoints := 8, Out.CamProfil[0].Status := 2, Out.CamProfil[1].Status := 2, Out.CamProfil[2].Status := 2, Out.CamProfil[3].Status := 2, Out.CamProfil[4].Status := 2, Out.CamProfil[5].Status := 2, Out.CamProfil[6].Status := 2, Out.CamProfil[7].Status := 2);
   PCAM_Inter_PCAM_Coupe_Fil : CAM[100] := ([0].SegmentType := 1, [1].Master := 180.0, [1].Slave := 90.0, [2].Master := 360.0, [2].Slave := 360.0, [2].SegmentType := 1);
   PCAM_Inter_PCAM_Horizontal : CAM[100] := ([1].Master := 1.0, [1].SegmentType := 1, [2].Master := 6.0, [2].Slave := 5.0, [3].Master := 36.0, [3].Slave := 77.0, [3].SegmentType := 1, [4].Master := 46.0, [4].Slave := 87.0, [5].Master := 51.0, [5].Slave := 87.0, [5].SegmentType := 1, [6].Master := 61.0, [6].Slave := 77.0, [6].SegmentType := 1, [7].Master := 90.0, [7].SegmentType := 1);
   PCAM_Inter_PCAM_Vertical : CAM[100] := ([0].Slave := 15.0, [1].Master := 1.0, [1].Slave := 15.0, [2].Master := 6.0, [2].Slave := 15.0, [3].Master := 48.0, [3].Slave := 15.0, [3].SegmentType := 1, [4].Master := 58.0, [4].Slave := 25.0, [5].Master := 63.0, [5].Slave := 25.0, [5].SegmentType := 1, [6].Master := 81.0, [6].Slave := 15.0, [7].Master := 90.0, [7].Slave := 15.0, [7].SegmentType := 1);
   PCAM_Vertical : UDT_CamGeneration := (Cmd.Start := 1, In.Cam[0].Slave := 15.0, In.Cam[1].Master := 1.0, In.Cam[1].Slave := 15.0, In.Cam[2].Master := 6.0, In.Cam[2].Slave := 15.0, In.Cam[3].Master := 48.0, In.Cam[3].Slave := 15.0, In.Cam[3].SegmentType := 1, In.Cam[4].Master := 58.0, In.Cam[4].Slave := 25.0, In.Cam[5].Master := 63.0, In.Cam[5].Slave := 25.0, In.Cam[5].SegmentType := 1, In.Cam[6].Master := 81.0, In.Cam[6].Slave := 15.0, In.Cam[7].Master := 90.0, In.Cam[7].Slave := 15.0, Out.Cam[0].Slave := 15.0, Out.Cam[1].Master := 1.0, Out.Cam[1].Slave := 15.0, Out.Cam[2].Master := 6.0, Out.Cam[2].Slave := 15.0, Out.Cam[3].Master := 48.0, Out.Cam[3].Slave := 15.0, Out.Cam[3].SegmentType := 1, Out.Cam[4].Master := 58.0, Out.Cam[4].Slave := 25.0, Out.Cam[5].Master := 63.0, Out.Cam[5].Slave := 25.0, Out.Cam[5].SegmentType := 1, Out.Cam[6].Master := 81.0, Out.Cam[6].Slave := 15.0, Out.Cam[7].Master := 90.0, Out.Cam[7].Slave := 15.0, Out.Cam[7].SegmentType := 1, Out.NbrOfCamPoints := 8, Out.CamProfil[0].Status := 2, Out.CamProfil[1].Status := 2, Out.CamProfil[2].Status := 2, Out.CamProfil[3].Status := 2, Out.CamProfil[4].Status := 2, Out.CamProfil[5].Status := 2, Out.CamProfil[6].Status := 2, Out.CamProfil[7].Status := 2);
   Periode_Top_Depart_Coupe_FIl : REAL := 1.875;
   Position_Codeur_Virtuel_Det_Produit : REAL := 59.0;
   Position_Codeur_Virtuel_Det_Produit_Moy : REAL := 66.833336;
   Position_Decalee : REAL := 52.0;
   Position_old_Tapis_Four : REAL := 9.62;
   Position_temp_Tapis_Four : REAL := 10.091;
   Raz_Axe_Coupe_Fil : Raz_Axe := (acc := 100000.0, dec := 100000.0, jerk := 1000000.0);
   Raz_Axe_H_Droit : Raz_Axe := (acc := 100000.0, dec := 100000.0, jerk := 1000000.0);
   Raz_Axe_H_Gauche : Raz_Axe := (acc := 100000.0, dec := 100000.0, jerk := 1000000.0);
   Raz_Axe_Pompe_Doseuse : Raz_Axe := (acc := 100000.0, dec := 100000.0, jerk := 1000000.0);
   Raz_Axe_Rouleaux : Raz_Axe := (acc := 100000.0, dec := 100000.0, jerk := 1000000.0);
   Raz_Axe_V_Droit : Raz_Axe := (acc := 100000.0, dec := 100000.0, jerk := 1000000.0);
   Raz_Axe_V_Gauche : Raz_Axe := (acc := 100000.0, dec := 100000.0, jerk := 1000000.0);
   RECETTE_CHAMP_VIDE : UDT_RECIPE;
   RECETTE_EC : UDT_RECIPE := (Name := 'SABLON 62x34 318SAB001', Comas.Pas_Machine := 90, Comas.Came_Maitre[1].Master := 90.0, Comas.Came_Maitre[1].Slave := 90.0, Comas.Longueur_Came_Maitre := 2, Comas.Tete.Stop_Cam_Logique_Degagement := 10.0, Comas.Tete.Position_Degagement_H := 50.0, Comas.Tete.Position_Degagement_V := 35.0, Comas.Tete.Hauteur_Tete := -14, Comas.Tete.Cam_Axe_Horizontal[1].Master := 1.0, Comas.Tete.Cam_Axe_Horizontal[1].SegmentType := 1, Comas.Tete.Cam_Axe_Horizontal[2].Master := 6.0, Comas.Tete.Cam_Axe_Horizontal[2].Slave := 5.0, Comas.Tete.Cam_Axe_Horizontal[3].Master := 36.0, Comas.Tete.Cam_Axe_Horizontal[3].Slave := 77.0, Comas.Tete.Cam_Axe_Horizontal[3].SegmentType := 1, Comas.Tete.Cam_Axe_Horizontal[4].Master := 46.0, Comas.Tete.Cam_Axe_Horizontal[4].Slave := 87.0, Comas.Tete.Cam_Axe_Horizontal[5].Master := 51.0, Comas.Tete.Cam_Axe_Horizontal[5].Slave := 87.0, Comas.Tete.Cam_Axe_Horizontal[5].SegmentType := 1, Comas.Tete.Cam_Axe_Horizontal[6].Master := 61.0, Comas.Tete.Cam_Axe_Horizontal[6].Slave := 77.0, Comas.Tete.Cam_Axe_Horizontal[6].SegmentType := 1, Comas.Tete.Cam_Axe_Horizontal[7].Master := 90.0, Comas.Tete.Cam_Axe_Vertical[0].Slave := 15.0, Comas.Tete.Cam_Axe_Vertical[1].Master := 1.0, Comas.Tete.Cam_Axe_Vertical[1].Slave := 15.0, Comas.Tete.Cam_Axe_Vertical[2].Master := 6.0, Comas.Tete.Cam_Axe_Vertical[2].Slave := 15.0, Comas.Tete.Cam_Axe_Vertical[3].Master := 48.0, Comas.Tete.Cam_Axe_Vertical[3].Slave := 15.0, Comas.Tete.Cam_Axe_Vertical[3].SegmentType := 1, Comas.Tete.Cam_Axe_Vertical[4].Master := 58.0, Comas.Tete.Cam_Axe_Vertical[4].Slave := 25.0, Comas.Tete.Cam_Axe_Vertical[5].Master := 63.0, Comas.Tete.Cam_Axe_Vertical[5].Slave := 25.0, Comas.Tete.Cam_Axe_Vertical[5].SegmentType := 1, Comas.Tete.Cam_Axe_Vertical[6].Master := 81.0, Comas.Tete.Cam_Axe_Vertical[6].Slave := 15.0, Comas.Tete.Cam_Axe_Vertical[7].Master := 90.0, Comas.Tete.Cam_Axe_Vertical[7].Slave := 15.0, Comas.Tete.Longueur_Cam_Axe_H := 8, Comas.Tete.Offset_Vertical_Gauche := 38.0, Comas.Tete.Offset_Horizontal_Gauche := 95.0, Comas.Tete.Cam_Axe_Horizontal_Pan.B.x := 1.0, Comas.Tete.Cam_Axe_Horizontal_Pan.C.x := 5.0, Comas.Tete.Cam_Axe_Horizontal_Pan.C.y := 5.0, Comas.Tete.Cam_Axe_Horizontal_Pan.D.x := 30.0, Comas.Tete.Cam_Axe_Horizontal_Pan.D.y := 75.0, Comas.Tete.Cam_Axe_Horizontal_Pan.E.x := 10.0, Comas.Tete.Cam_Axe_Horizontal_Pan.E.y := 10.0, Comas.Tete.Cam_Axe_Horizontal_Pan.F.x := 5.0, Comas.Tete.Cam_Axe_Horizontal_Pan.G.x := 10.0, Comas.Tete.Cam_Axe_Horizontal_Pan.G.y := -10.0, Comas.Tete.Cam_Axe_Vertical_Pan.H.y := 15.0, Comas.Tete.Cam_Axe_Vertical_Pan.I.y := 15.0, Comas.Tete.Cam_Axe_Vertical_Pan.J.y := 15.0, Comas.Tete.Cam_Axe_Vertical_Pan.K.x := 12.0, Comas.Tete.Cam_Axe_Vertical_Pan.K.y := 15.0,
        Comas.Tete.Cam_Axe_Vertical_Pan.L.x := 12.0, Comas.Tete.Cam_Axe_Vertical_Pan.L.y := 25.0, Comas.Tete.Cam_Axe_Vertical_Pan.M.x := 12.0, Comas.Tete.Cam_Axe_Vertical_Pan.M.y := 25.0, Comas.Tete.Cam_Axe_Vertical_Pan.N.x := 20.0, Comas.Tete.Cam_Axe_Vertical_Pan.N.y := 15.0, Comas.Tete.Offset_Vertical_Droit := 45.0, Comas.Tete.Offset_Horizontal_Droit := 95.0, Comas.Tete.Reserve_Real1 := -3.0, Comas.Pompe.Start_Cam_Logique_Avance := -19.0, Comas.Pompe.Stop_Cam_Logique_Avance := 31.0, Comas.Pompe.Start_Cam_Logique_Recul := 43.0, Comas.Pompe.Stop_Cam_Logique_Recul := 63.0, Comas.Pompe.Consigne_Vitesse_Avance := 11.2, Comas.Pompe.Consigne_Acc_Dec_Avance := 40.0, Comas.Pompe.Consigne_Jerk_Avance := 100.0, Comas.Pompe.Consigne_Vitesse_Recul := -10.0, Comas.Pompe.Consigne_Acc_Dec_Recul := 40.0, Comas.Pompe.Consigne_Jerk_Recul := 100.0, Comas.Pompe.Points_Pan.O.x := -25.0, Comas.Pompe.Points_Pan.Q.x := 50.0, Comas.Pompe.Points_Pan.S.x := -5.0, Comas.Pompe.Points_Pan.U.x := 20.0, Comas.Pompe.Reserve_Bool1 := 1, Comas.Rouleaux.Syncho_Pompe := 1, Comas.Rouleaux.Consigne_Vitesse := 25.0, Comas.Rouleaux.Consigne_Acc_Dec := 40.0, Comas.Rouleaux.Consigne_Jerk := 100.0, Comas.Coupe_Fil.Start_Cam_Logique_Virtuelle := 11.0, Comas.Coupe_Fil.Stop_Cam_Logique_Virtuelle := 21.0, Comas.Coupe_Fil.Consigne_Vitesse_Virtuelle := 200.0, Comas.Coupe_Fil.Consigne_Acc_Dec_Virtuelle := 1000.0, Comas.Coupe_Fil.Consigne_Jerk_Virtuelle := 50.0, Comas.Coupe_Fil.Cam_Axe[0].SegmentType := 1, Comas.Coupe_Fil.Cam_Axe[1].Master := 180.0, Comas.Coupe_Fil.Cam_Axe[1].Slave := 90.0, Comas.Coupe_Fil.Cam_Axe[2].Master := 360.0, Comas.Coupe_Fil.Cam_Axe[2].Slave := 360.0, Comas.Coupe_Fil.Cam_Axe[2].SegmentType := 1, Comas.Coupe_Fil.Points_Pan.W.x := 30.0, Comas.Consigne_Vitesse_Manu_mm := 2.0, Comas.Consigne_Acc_Decc_Manu_mm := 10.0, Comas.Consigne_Jerk_Manu := 100.0, Comas.Activation_Cam_Auto := 1, Comas.Distance_CPT_Presence_Produit := 520, Comas.Consigne_Vitesse_Manu_Tour := 10.0, Comas.Consigne_Acc_Decc_Manu_Tour := 10.0, Comas.Mode_Decoreuse_Cam_Logique := 1, Comas.Reserve_Real3 := 1.0, Comas.Reserve_Real4 := 1.0, Comas.Reserve_Real5 := 5.0, Reserve_Real2 := 200.0, Reserve_Real3 := 10.0);
   RECETTE_HMI : UDT_HMI := (Index_Recette_a_supprimer := 3);
   RECETTE_SV : UDT_RECIPE[50] := ([0].Name := 'SABLON 62x34 318SAB001', [0].Comas.Pas_Machine := 90, [0].Comas.Came_Maitre[1].Master := 90.0, [0].Comas.Came_Maitre[1].Slave := 90.0, [0].Comas.Longueur_Came_Maitre := 2, [0].Comas.Tete.Stop_Cam_Logique_Degagement := 10.0, [0].Comas.Tete.Position_Degagement_H := 50.0, [0].Comas.Tete.Position_Degagement_V := 35.0, [0].Comas.Tete.Hauteur_Tete := -5, [0].Comas.Tete.Cam_Axe_Horizontal[1].Master := 1.0, [0].Comas.Tete.Cam_Axe_Horizontal[1].SegmentType := 1, [0].Comas.Tete.Cam_Axe_Horizontal[2].Master := 6.0, [0].Comas.Tete.Cam_Axe_Horizontal[2].Slave := 5.0, [0].Comas.Tete.Cam_Axe_Horizontal[3].Master := 36.0, [0].Comas.Tete.Cam_Axe_Horizontal[3].Slave := 78.0, [0].Comas.Tete.Cam_Axe_Horizontal[3].SegmentType := 1, [0].Comas.Tete.Cam_Axe_Horizontal[4].Master := 46.0, [0].Comas.Tete.Cam_Axe_Horizontal[4].Slave := 88.0, [0].Comas.Tete.Cam_Axe_Horizontal[5].Master := 51.0, [0].Comas.Tete.Cam_Axe_Horizontal[5].Slave := 88.0, [0].Comas.Tete.Cam_Axe_Horizontal[5].SegmentType := 1, [0].Comas.Tete.Cam_Axe_Horizontal[6].Master := 61.0, [0].Comas.Tete.Cam_Axe_Horizontal[6].Slave := 78.0, [0].Comas.Tete.Cam_Axe_Horizontal[6].SegmentType := 1, [0].Comas.Tete.Cam_Axe_Horizontal[7].Master := 90.0, [0].Comas.Tete.Cam_Axe_Vertical[0].Slave := 15.0, [0].Comas.Tete.Cam_Axe_Vertical[1].Master := 1.0, [0].Comas.Tete.Cam_Axe_Vertical[1].Slave := 15.0, [0].Comas.Tete.Cam_Axe_Vertical[2].Master := 6.0, [0].Comas.Tete.Cam_Axe_Vertical[2].Slave := 15.0, [0].Comas.Tete.Cam_Axe_Vertical[3].Master := 48.0, [0].Comas.Tete.Cam_Axe_Vertical[3].Slave := 15.0, [0].Comas.Tete.Cam_Axe_Vertical[3].SegmentType := 1, [0].Comas.Tete.Cam_Axe_Vertical[4].Master := 58.0, [0].Comas.Tete.Cam_Axe_Vertical[4].Slave := 25.0, [0].Comas.Tete.Cam_Axe_Vertical[5].Master := 63.0, [0].Comas.Tete.Cam_Axe_Vertical[5].Slave := 25.0, [0].Comas.Tete.Cam_Axe_Vertical[5].SegmentType := 1, [0].Comas.Tete.Cam_Axe_Vertical[6].Master := 81.0, [0].Comas.Tete.Cam_Axe_Vertical[6].Slave := 15.0, [0].Comas.Tete.Cam_Axe_Vertical[7].Master := 90.0, [0].Comas.Tete.Cam_Axe_Vertical[7].Slave := 15.0, [0].Comas.Tete.Longueur_Cam_Axe_H := 8, [0].Comas.Tete.Offset_Vertical_Gauche := 38.0, [0].Comas.Tete.Offset_Horizontal_Gauche := 95.0, [0].Comas.Tete.Cam_Axe_Horizontal_Pan.B.x := 1.0, [0].Comas.Tete.Cam_Axe_Horizontal_Pan.C.x := 5.0, [0].Comas.Tete.Cam_Axe_Horizontal_Pan.C.y := 5.0, [0].Comas.Tete.Cam_Axe_Horizontal_Pan.D.x := 30.0, [0].Comas.Tete.Cam_Axe_Horizontal_Pan.D.y := 75.0, [0].Comas.Tete.Cam_Axe_Horizontal_Pan.E.x := 10.0, [0].Comas.Tete.Cam_Axe_Horizontal_Pan.E.y := 10.0, [0].Comas.Tete.Cam_Axe_Horizontal_Pan.F.x := 5.0, [0].Comas.Tete.Cam_Axe_Horizontal_Pan.G.x := 10.0, [0].Comas.Tete.Cam_Axe_Horizontal_Pan.G.y := -10.0, [0].Comas.Tete.Cam_Axe_Vertical_Pan.H.y := 15.0, [0].Comas.Tete.Cam_Axe_Vertical_Pan.I.y := 15.0, [0].Comas.Tete.Cam_Axe_Vertical_Pan.J.y := 15.0, [0].Comas.Tete.Cam_Axe_Vertical_Pan.K.x := 12.0, [0].Comas.Tete.Cam_Axe_Vertical_Pan.K.y := 15.0,
        [0].Comas.Tete.Cam_Axe_Vertical_Pan.L.x := 12.0, [0].Comas.Tete.Cam_Axe_Vertical_Pan.L.y := 25.0, [0].Comas.Tete.Cam_Axe_Vertical_Pan.M.x := 12.0, [0].Comas.Tete.Cam_Axe_Vertical_Pan.M.y := 25.0, [0].Comas.Tete.Cam_Axe_Vertical_Pan.N.x := 20.0, [0].Comas.Tete.Cam_Axe_Vertical_Pan.N.y := 15.0, [0].Comas.Tete.Offset_Vertical_Droit := 45.0, [0].Comas.Tete.Offset_Horizontal_Droit := 95.0, [0].Comas.Tete.Reserve_Real1 := -2.0, [0].Comas.Pompe.Start_Cam_Logique_Avance := -19.0, [0].Comas.Pompe.Stop_Cam_Logique_Avance := 31.0, [0].Comas.Pompe.Start_Cam_Logique_Recul := 43.0, [0].Comas.Pompe.Stop_Cam_Logique_Recul := 63.0, [0].Comas.Pompe.Consigne_Vitesse_Avance := 11.0, [0].Comas.Pompe.Consigne_Acc_Dec_Avance := 40.0, [0].Comas.Pompe.Consigne_Jerk_Avance := 100.0, [0].Comas.Pompe.Consigne_Vitesse_Recul := -10.0, [0].Comas.Pompe.Consigne_Acc_Dec_Recul := 40.0, [0].Comas.Pompe.Consigne_Jerk_Recul := 100.0, [0].Comas.Pompe.Points_Pan.O.x := -25.0, [0].Comas.Pompe.Points_Pan.Q.x := 50.0, [0].Comas.Pompe.Points_Pan.S.x := -5.0, [0].Comas.Pompe.Points_Pan.U.x := 20.0, [0].Comas.Pompe.Reserve_Bool1 := 1, [0].Comas.Rouleaux.Syncho_Pompe := 1, [0].Comas.Rouleaux.Consigne_Vitesse := 25.0, [0].Comas.Rouleaux.Consigne_Acc_Dec := 40.0, [0].Comas.Rouleaux.Consigne_Jerk := 100.0, [0].Comas.Coupe_Fil.Start_Cam_Logique_Virtuelle := 11.0, [0].Comas.Coupe_Fil.Stop_Cam_Logique_Virtuelle := 21.0, [0].Comas.Coupe_Fil.Consigne_Vitesse_Virtuelle := 200.0, [0].Comas.Coupe_Fil.Consigne_Acc_Dec_Virtuelle := 1000.0, [0].Comas.Coupe_Fil.Consigne_Jerk_Virtuelle := 50.0, [0].Comas.Coupe_Fil.Cam_Axe[0].SegmentType := 1, [0].Comas.Coupe_Fil.Cam_Axe[1].Master := 180.0, [0].Comas.Coupe_Fil.Cam_Axe[1].Slave := 90.0, [0].Comas.Coupe_Fil.Cam_Axe[2].Master := 360.0, [0].Comas.Coupe_Fil.Cam_Axe[2].Slave := 360.0, [0].Comas.Coupe_Fil.Cam_Axe[2].SegmentType := 1, [0].Comas.Coupe_Fil.Points_Pan.W.x := 30.0, [0].Comas.Consigne_Vitesse_Manu_mm := 2.0, [0].Comas.Consigne_Acc_Decc_Manu_mm := 10.0, [0].Comas.Consigne_Jerk_Manu := 100.0, [0].Comas.Activation_Cam_Auto := 1, [0].Comas.Distance_CPT_Presence_Produit := 520, [0].Comas.Consigne_Vitesse_Manu_Tour := 10.0, [0].Comas.Consigne_Acc_Decc_Manu_Tour := 10.0, [0].Comas.Mode_Decoreuse_Cam_Logique := 1, [1].Name := 'MERINGUE CARRE', [1].Comas.Pas_Machine := 54, [1].Comas.Came_Maitre[1].Master := 54.0, [1].Comas.Came_Maitre[1].Slave := 54.0, [1].Comas.Longueur_Came_Maitre := 2, [1].Comas.Tete.Stop_Cam_Logique_Degagement := 10.0, [1].Comas.Tete.Position_Degagement_H := 50.0, [1].Comas.Tete.Position_Degagement_V := 35.0, [1].Comas.Tete.Hauteur_Tete := 6, [1].Comas.Tete.Cam_Axe_Horizontal[1].Master := 1.0, [1].Comas.Tete.Cam_Axe_Horizontal[1].SegmentType := 1, [1].Comas.Tete.Cam_Axe_Horizontal[2].Master := 6.0,
        [1].Comas.Tete.Cam_Axe_Horizontal[2].Slave := 2.0, [1].Comas.Tete.Cam_Axe_Horizontal[3].Master := 21.0, [1].Comas.Tete.Cam_Axe_Horizontal[3].Slave := 30.0, [1].Comas.Tete.Cam_Axe_Horizontal[3].SegmentType := 1, [1].Comas.Tete.Cam_Axe_Horizontal[4].Master := 26.0, [1].Comas.Tete.Cam_Axe_Horizontal[4].Slave := 35.0, [1].Comas.Tete.Cam_Axe_Horizontal[5].Master := 34.0, [1].Comas.Tete.Cam_Axe_Horizontal[5].Slave := 35.0, [1].Comas.Tete.Cam_Axe_Horizontal[5].SegmentType := 1, [1].Comas.Tete.Cam_Axe_Horizontal[6].Master := 44.0, [1].Comas.Tete.Cam_Axe_Horizontal[6].Slave := 25.0, [1].Comas.Tete.Cam_Axe_Horizontal[6].SegmentType := 1, [1].Comas.Tete.Cam_Axe_Horizontal[7].Master := 54.0, [1].Comas.Tete.Cam_Axe_Vertical[1].Master := 1.0, [1].Comas.Tete.Cam_Axe_Vertical[2].Master := 6.0, [1].Comas.Tete.Cam_Axe_Vertical[3].Master := 21.0, [1].Comas.Tete.Cam_Axe_Vertical[3].SegmentType := 1, [1].Comas.Tete.Cam_Axe_Vertical[4].Master := 31.0, [1].Comas.Tete.Cam_Axe_Vertical[4].Slave := 5.0, [1].Comas.Tete.Cam_Axe_Vertical[5].Master := 39.0, [1].Comas.Tete.Cam_Axe_Vertical[5].Slave := 5.0, [1].Comas.Tete.Cam_Axe_Vertical[5].SegmentType := 1, [1].Comas.Tete.Cam_Axe_Vertical[6].Master := 52.0, [1].Comas.Tete.Cam_Axe_Vertical[7].Master := 54.0, [1].Comas.Tete.Longueur_Cam_Axe_H := 8, [1].Comas.Tete.Offset_Vertical_Gauche := 38.0, [1].Comas.Tete.Offset_Horizontal_Gauche := 95.0, [1].Comas.Tete.Cam_Axe_Horizontal_Pan.B.x := 1.0, [1].Comas.Tete.Cam_Axe_Horizontal_Pan.C.x := 5.0, [1].Comas.Tete.Cam_Axe_Horizontal_Pan.C.y := 2.0, [1].Comas.Tete.Cam_Axe_Horizontal_Pan.D.x := 15.0, [1].Comas.Tete.Cam_Axe_Horizontal_Pan.D.y := 25.0, [1].Comas.Tete.Cam_Axe_Horizontal_Pan.E.x := 5.0, [1].Comas.Tete.Cam_Axe_Horizontal_Pan.E.y := 5.0, [1].Comas.Tete.Cam_Axe_Horizontal_Pan.F.x := 8.0, [1].Comas.Tete.Cam_Axe_Horizontal_Pan.G.x := 10.0, [1].Comas.Tete.Cam_Axe_Horizontal_Pan.G.y := -10.0, [1].Comas.Tete.Cam_Axe_Vertical_Pan.L.x := 5.0, [1].Comas.Tete.Cam_Axe_Vertical_Pan.L.y := 5.0, [1].Comas.Tete.Cam_Axe_Vertical_Pan.M.x := 5.0, [1].Comas.Tete.Cam_Axe_Vertical_Pan.M.y := 5.0, [1].Comas.Tete.Cam_Axe_Vertical_Pan.N.x := 8.0, [1].Comas.Tete.Offset_Vertical_Droit := 45.0, [1].Comas.Tete.Offset_Horizontal_Droit := 95.0, [1].Comas.Tete.Reserve_Real1 := 3.0, [1].Comas.Pompe.Start_Cam_Logique_Avance := -14.0, [1].Comas.Pompe.Stop_Cam_Logique_Avance := 16.0, [1].Comas.Pompe.Start_Cam_Logique_Recul := 16.0, [1].Comas.Pompe.Stop_Cam_Logique_Recul := 36.0, [1].Comas.Pompe.Consigne_Vitesse_Avance := 21.2, [1].Comas.Pompe.Consigne_Acc_Dec_Avance := 40.0, [1].Comas.Pompe.Consigne_Jerk_Avance := 100.0, [1].Comas.Pompe.Consigne_Vitesse_Recul := -20.5, [1].Comas.Pompe.Consigne_Acc_Dec_Recul := 40.0, [1].Comas.Pompe.Consigne_Jerk_Recul := 100.0, [1].Comas.Pompe.Points_Pan.O.x := -20.0, [1].Comas.Pompe.Points_Pan.Q.x := 30.0, [1].Comas.Pompe.Points_Pan.S.x := -5.0, [1].Comas.Pompe.Points_Pan.U.x := 20.0, [1].Comas.Pompe.Reserve_Bool1 := 1,
        [1].Comas.Rouleaux.Syncho_Pompe := 1, [1].Comas.Rouleaux.Consigne_Vitesse := 19.5, [1].Comas.Rouleaux.Consigne_Acc_Dec := 40.0, [1].Comas.Rouleaux.Consigne_Jerk := 100.0, [1].Comas.Coupe_Fil.Start_Cam_Logique_Virtuelle := 16.0, [1].Comas.Coupe_Fil.Stop_Cam_Logique_Virtuelle := 26.0, [1].Comas.Coupe_Fil.Consigne_Vitesse_Virtuelle := 200.0, [1].Comas.Coupe_Fil.Consigne_Acc_Dec_Virtuelle := 1000.0, [1].Comas.Coupe_Fil.Consigne_Jerk_Virtuelle := 50.0, [1].Comas.Coupe_Fil.Cam_Axe[0].SegmentType := 1, [1].Comas.Coupe_Fil.Cam_Axe[1].Master := 180.0, [1].Comas.Coupe_Fil.Cam_Axe[1].Slave := 90.0, [1].Comas.Coupe_Fil.Cam_Axe[2].Master := 360.0, [1].Comas.Coupe_Fil.Cam_Axe[2].Slave := 360.0, [1].Comas.Coupe_Fil.Cam_Axe[2].SegmentType := 1, [1].Comas.Coupe_Fil.Points_Pan.W.x := 30.0, [1].Comas.Consigne_Vitesse_Manu_mm := 2.0, [1].Comas.Consigne_Acc_Decc_Manu_mm := 10.0, [1].Comas.Consigne_Jerk_Manu := 100.0, [1].Comas.Activation_Cam_Auto := 1, [1].Comas.Distance_CPT_Presence_Produit := 520, [1].Comas.Consigne_Vitesse_Manu_Tour := 10.0, [1].Comas.Consigne_Acc_Decc_Manu_Tour := 10.0, [1].Comas.Reserve_Real3 := 1.0, [1].Comas.Reserve_Real4 := 1.0, [1].Comas.Reserve_Real5 := 5.0, [1].Comas.Reserve_Real6 := 200.0, [1].Reserve_Real2 := 200.0, [1].Reserve_Real3 := 10.0, [2].Name := 'COOKIE 311MIN011', [2].Comas.Pas_Machine := 95, [2].Comas.Came_Maitre[1].Master := 95.0, [2].Comas.Came_Maitre[1].Slave := 95.0, [2].Comas.Longueur_Came_Maitre := 2, [2].Comas.Tete.Stop_Cam_Logique_Degagement := 10.0, [2].Comas.Tete.Position_Degagement_H := 50.0, [2].Comas.Tete.Position_Degagement_V := 35.0, [2].Comas.Tete.Cam_Axe_Horizontal[1].Master := 1.0, [2].Comas.Tete.Cam_Axe_Horizontal[1].SegmentType := 1, [2].Comas.Tete.Cam_Axe_Horizontal[2].Master := 11.0, [2].Comas.Tete.Cam_Axe_Horizontal[2].Slave := 5.0, [2].Comas.Tete.Cam_Axe_Horizontal[3].Master := 41.0, [2].Comas.Tete.Cam_Axe_Horizontal[3].Slave := 35.0, [2].Comas.Tete.Cam_Axe_Horizontal[3].SegmentType := 1, [2].Comas.Tete.Cam_Axe_Horizontal[4].Master := 51.0, [2].Comas.Tete.Cam_Axe_Horizontal[4].Slave := 40.0, [2].Comas.Tete.Cam_Axe_Horizontal[5].Master := 61.0, [2].Comas.Tete.Cam_Axe_Horizontal[5].Slave := 40.0, [2].Comas.Tete.Cam_Axe_Horizontal[5].SegmentType := 1, [2].Comas.Tete.Cam_Axe_Horizontal[6].Master := 71.0, [2].Comas.Tete.Cam_Axe_Horizontal[6].Slave := 30.0, [2].Comas.Tete.Cam_Axe_Horizontal[6].SegmentType := 1, [2].Comas.Tete.Cam_Axe_Horizontal[7].Master := 95.0, [2].Comas.Tete.Cam_Axe_Vertical[1].Master := 1.0, [2].Comas.Tete.Cam_Axe_Vertical[2].Master := 11.0, [2].Comas.Tete.Cam_Axe_Vertical[3].Master := 41.0, [2].Comas.Tete.Cam_Axe_Vertical[3].SegmentType := 1, [2].Comas.Tete.Cam_Axe_Vertical[4].Master := 56.0, [2].Comas.Tete.Cam_Axe_Vertical[4].Slave := 10.0, [2].Comas.Tete.Cam_Axe_Vertical[5].Master := 66.0,
        [2].Comas.Tete.Cam_Axe_Vertical[5].Slave := 10.0, [2].Comas.Tete.Cam_Axe_Vertical[5].SegmentType := 1, [2].Comas.Tete.Cam_Axe_Vertical[6].Master := 86.0, [2].Comas.Tete.Cam_Axe_Vertical[7].Master := 95.0, [2].Comas.Tete.Longueur_Cam_Axe_H := 8, [2].Comas.Tete.Offset_Vertical_Gauche := 38.0, [2].Comas.Tete.Offset_Horizontal_Gauche := 95.0, [2].Comas.Tete.Cam_Axe_Horizontal_Pan.B.x := 1.0, [2].Comas.Tete.Cam_Axe_Horizontal_Pan.C.x := 10.0, [2].Comas.Tete.Cam_Axe_Horizontal_Pan.C.y := 5.0, [2].Comas.Tete.Cam_Axe_Horizontal_Pan.D.x := 30.0, [2].Comas.Tete.Cam_Axe_Horizontal_Pan.D.y := 30.0, [2].Comas.Tete.Cam_Axe_Horizontal_Pan.E.x := 10.0, [2].Comas.Tete.Cam_Axe_Horizontal_Pan.E.y := 5.0, [2].Comas.Tete.Cam_Axe_Horizontal_Pan.F.x := 10.0, [2].Comas.Tete.Cam_Axe_Horizontal_Pan.G.x := 10.0, [2].Comas.Tete.Cam_Axe_Horizontal_Pan.G.y := -10.0, [2].Comas.Tete.Cam_Axe_Vertical_Pan.L.x := 5.0, [2].Comas.Tete.Cam_Axe_Vertical_Pan.L.y := 10.0, [2].Comas.Tete.Cam_Axe_Vertical_Pan.M.x := 5.0, [2].Comas.Tete.Cam_Axe_Vertical_Pan.M.y := 10.0, [2].Comas.Tete.Cam_Axe_Vertical_Pan.N.x := 15.0, [2].Comas.Tete.Offset_Vertical_Droit := 45.0, [2].Comas.Tete.Offset_Horizontal_Droit := 95.0, [2].Comas.Pompe.Start_Cam_Logique_Avance := 1.0, [2].Comas.Pompe.Stop_Cam_Logique_Avance := 14.0, [2].Comas.Pompe.Start_Cam_Logique_Recul := 41.0, [2].Comas.Pompe.Stop_Cam_Logique_Recul := 41.0, [2].Comas.Pompe.Consigne_Vitesse_Avance := 13.5, [2].Comas.Pompe.Consigne_Acc_Dec_Avance := 40.0, [2].Comas.Pompe.Consigne_Jerk_Avance := 100.0, [2].Comas.Pompe.Consigne_Acc_Dec_Recul := 40.0, [2].Comas.Pompe.Consigne_Jerk_Recul := 100.0, [2].Comas.Pompe.Points_Pan.O.x := -10.0, [2].Comas.Pompe.Points_Pan.Q.x := 13.0, [2].Comas.Pompe.Reserve_Bool1 := 1, [2].Comas.Rouleaux.Syncho_Pompe := 1, [2].Comas.Rouleaux.Consigne_Vitesse := 31.0, [2].Comas.Rouleaux.Consigne_Acc_Dec := 40.0, [2].Comas.Rouleaux.Consigne_Jerk := 100.0, [2].Comas.Coupe_Fil.Activation := 1, [2].Comas.Coupe_Fil.Start_Cam_Logique_Virtuelle := 11.0, [2].Comas.Coupe_Fil.Stop_Cam_Logique_Virtuelle := 21.0, [2].Comas.Coupe_Fil.Consigne_Vitesse_Virtuelle := 250.0, [2].Comas.Coupe_Fil.Consigne_Acc_Dec_Virtuelle := 1000.0, [2].Comas.Coupe_Fil.Consigne_Jerk_Virtuelle := 50.0, [2].Comas.Coupe_Fil.Cam_Axe[0].SegmentType := 1, [2].Comas.Coupe_Fil.Cam_Axe[1].Master := 180.0, [2].Comas.Coupe_Fil.Cam_Axe[1].Slave := 180.0, [2].Comas.Coupe_Fil.Cam_Axe[2].Master := 250.0, [2].Comas.Coupe_Fil.Cam_Axe[2].Slave := 180.0, [2].Comas.Coupe_Fil.Cam_Axe[2].SegmentType := 1, [2].Comas.Coupe_Fil.Cam_Axe[3].Master := 360.0, [2].Comas.Coupe_Fil.Cam_Axe[3].Slave := 360.0, [2].Comas.Coupe_Fil.Cam_Axe[3].SegmentType := 1, [2].Comas.Coupe_Fil.Cam_Axe[4].SegmentType := 1, [2].Comas.Coupe_Fil.Points_Pan.W.x := -40.0, [2].Comas.Coupe_Fil.Reserve_Bool1 := 1, [2].Comas.Consigne_Vitesse_Manu_mm := 2.0, [2].Comas.Consigne_Acc_Decc_Manu_mm := 10.0,
        [2].Comas.Consigne_Jerk_Manu := 100.0, [2].Comas.Activation_Cam_Auto := 1, [2].Comas.Distance_CPT_Presence_Produit := 520, [2].Comas.Consigne_Vitesse_Manu_Tour := 10.0, [2].Comas.Consigne_Acc_Decc_Manu_Tour := 10.0, [2].Comas.Mode_Decoreuse_Cam_Logique := 1, [2].Comas.Reserve_Real6 := 200.0, [4].Name := 'Sablon MDLZ', [4].Comas.Pas_Machine := 60, [4].Comas.Came_Maitre[1].Master := 60.0, [4].Comas.Came_Maitre[1].Slave := 60.0, [4].Comas.Longueur_Came_Maitre := 2, [4].Comas.Tete.Stop_Cam_Logique_Degagement := 10.0, [4].Comas.Tete.Position_Degagement_H := 50.0, [4].Comas.Tete.Position_Degagement_V := 35.0, [4].Comas.Tete.Hauteur_Tete := -12, [4].Comas.Tete.Cam_Axe_Horizontal[1].Master := 1.0, [4].Comas.Tete.Cam_Axe_Horizontal[1].SegmentType := 1, [4].Comas.Tete.Cam_Axe_Horizontal[2].Master := 6.0, [4].Comas.Tete.Cam_Axe_Horizontal[2].Slave := 2.0, [4].Comas.Tete.Cam_Axe_Horizontal[3].Master := 21.0, [4].Comas.Tete.Cam_Axe_Horizontal[3].Slave := 22.0, [4].Comas.Tete.Cam_Axe_Horizontal[3].SegmentType := 1, [4].Comas.Tete.Cam_Axe_Horizontal[4].Master := 31.0, [4].Comas.Tete.Cam_Axe_Horizontal[4].Slave := 27.0, [4].Comas.Tete.Cam_Axe_Horizontal[5].Master := 36.0, [4].Comas.Tete.Cam_Axe_Horizontal[5].Slave := 27.0, [4].Comas.Tete.Cam_Axe_Horizontal[5].SegmentType := 1, [4].Comas.Tete.Cam_Axe_Horizontal[6].Master := 46.0, [4].Comas.Tete.Cam_Axe_Horizontal[6].Slave := 27.0, [4].Comas.Tete.Cam_Axe_Horizontal[6].SegmentType := 1, [4].Comas.Tete.Cam_Axe_Horizontal[7].Master := 60.0, [4].Comas.Tete.Cam_Axe_Vertical[1].Master := 1.0, [4].Comas.Tete.Cam_Axe_Vertical[2].Master := 6.0, [4].Comas.Tete.Cam_Axe_Vertical[3].Master := 11.0, [4].Comas.Tete.Cam_Axe_Vertical[3].SegmentType := 1, [4].Comas.Tete.Cam_Axe_Vertical[4].Master := 21.0, [4].Comas.Tete.Cam_Axe_Vertical[4].Slave := 5.0, [4].Comas.Tete.Cam_Axe_Vertical[5].Master := 41.0, [4].Comas.Tete.Cam_Axe_Vertical[5].Slave := 9.0, [4].Comas.Tete.Cam_Axe_Vertical[5].SegmentType := 1, [4].Comas.Tete.Cam_Axe_Vertical[6].Master := 56.0, [4].Comas.Tete.Cam_Axe_Vertical[7].Master := 60.0, [4].Comas.Tete.Longueur_Cam_Axe_H := 8, [4].Comas.Tete.Offset_Vertical_Gauche := 38.0, [4].Comas.Tete.Offset_Horizontal_Gauche := 95.0, [4].Comas.Tete.Cam_Axe_Horizontal_Pan.B.x := 1.0, [4].Comas.Tete.Cam_Axe_Horizontal_Pan.C.x := 5.0, [4].Comas.Tete.Cam_Axe_Horizontal_Pan.C.y := 2.0, [4].Comas.Tete.Cam_Axe_Horizontal_Pan.D.x := 15.0, [4].Comas.Tete.Cam_Axe_Horizontal_Pan.D.y := 28.0, [4].Comas.Tete.Cam_Axe_Horizontal_Pan.E.x := 10.0, [4].Comas.Tete.Cam_Axe_Horizontal_Pan.E.y := 5.0, [4].Comas.Tete.Cam_Axe_Horizontal_Pan.F.x := 5.0, [4].Comas.Tete.Cam_Axe_Horizontal_Pan.G.x := 10.0, [4].Comas.Tete.Cam_Axe_Vertical_Pan.K.x := -10.0, [4].Comas.Tete.Cam_Axe_Vertical_Pan.L.x := -10.0, [4].Comas.Tete.Cam_Axe_Vertical_Pan.L.y := 5.0, [4].Comas.Tete.Cam_Axe_Vertical_Pan.M.x := 5.0, [4].Comas.Tete.Cam_Axe_Vertical_Pan.M.y := 9.0,
        [4].Comas.Tete.Cam_Axe_Vertical_Pan.N.x := 10.0, [4].Comas.Tete.Offset_Vertical_Droit := 45.0, [4].Comas.Tete.Offset_Horizontal_Droit := 95.0, [4].Comas.Tete.Reserve_Real1 := -8.0, [4].Comas.Pompe.Start_Cam_Logique_Avance := -8.0, [4].Comas.Pompe.Stop_Cam_Logique_Avance := 7.0, [4].Comas.Pompe.Start_Cam_Logique_Recul := 7.0, [4].Comas.Pompe.Stop_Cam_Logique_Recul := 22.0, [4].Comas.Pompe.Consigne_Vitesse_Avance := 47.5, [4].Comas.Pompe.Consigne_Acc_Dec_Avance := 40.0, [4].Comas.Pompe.Consigne_Jerk_Avance := 100.0, [4].Comas.Pompe.Consigne_Vitesse_Recul := -28.0, [4].Comas.Pompe.Consigne_Acc_Dec_Recul := 40.0, [4].Comas.Pompe.Consigne_Jerk_Recul := 100.0, [4].Comas.Pompe.Points_Pan.O.x := -14.0, [4].Comas.Pompe.Points_Pan.Q.x := 15.0, [4].Comas.Pompe.Points_Pan.S.x := -4.0, [4].Comas.Pompe.Points_Pan.U.x := 15.0, [4].Comas.Pompe.Reserve_Bool1 := 1, [4].Comas.Rouleaux.Consigne_Vitesse := 25.0, [4].Comas.Rouleaux.Consigne_Acc_Dec := 40.0, [4].Comas.Rouleaux.Consigne_Jerk := 100.0, [4].Comas.Rouleaux.Reserve_Real1 := -15.0, [4].Comas.Coupe_Fil.Start_Cam_Logique_Virtuelle := 11.0, [4].Comas.Coupe_Fil.Stop_Cam_Logique_Virtuelle := 21.0, [4].Comas.Coupe_Fil.Consigne_Vitesse_Virtuelle := 200.0, [4].Comas.Coupe_Fil.Consigne_Acc_Dec_Virtuelle := 1000.0, [4].Comas.Coupe_Fil.Consigne_Jerk_Virtuelle := 50.0, [4].Comas.Coupe_Fil.Cam_Axe[0].SegmentType := 1, [4].Comas.Coupe_Fil.Cam_Axe[1].Master := 180.0, [4].Comas.Coupe_Fil.Cam_Axe[1].Slave := 90.0, [4].Comas.Coupe_Fil.Cam_Axe[2].Master := 360.0, [4].Comas.Coupe_Fil.Cam_Axe[2].Slave := 360.0, [4].Comas.Coupe_Fil.Cam_Axe[2].SegmentType := 1, [4].Comas.Coupe_Fil.Points_Pan.W.x := 30.0, [4].Comas.Consigne_Vitesse_Manu_mm := 4.0, [4].Comas.Consigne_Acc_Decc_Manu_mm := 10.0, [4].Comas.Consigne_Jerk_Manu := 100.0, [4].Comas.Activation_Cam_Auto := 1, [4].Comas.Distance_CPT_Presence_Produit := 520, [4].Comas.Consigne_Vitesse_Manu_Tour := 10.0, [4].Comas.Consigne_Acc_Decc_Manu_Tour := 10.0, [4].Comas.Mode_Decoreuse_Cam_Logique := 1, [4].Comas.Reserve_Real6 := 200.0, [5].Name := 'LANGUE 40', [5].Comas.Pas_Machine := 70, [5].Comas.Came_Maitre[1].Master := 70.0, [5].Comas.Came_Maitre[1].Slave := 70.0, [5].Comas.Longueur_Came_Maitre := 2, [5].Comas.Tete.Stop_Cam_Logique_Degagement := 10.0, [5].Comas.Tete.Position_Degagement_H := 50.0, [5].Comas.Tete.Position_Degagement_V := 35.0, [5].Comas.Tete.Hauteur_Tete := -2, [5].Comas.Tete.Cam_Axe_Horizontal[1].Master := 1.0, [5].Comas.Tete.Cam_Axe_Horizontal[1].SegmentType := 1, [5].Comas.Tete.Cam_Axe_Horizontal[2].Master := 6.0, [5].Comas.Tete.Cam_Axe_Horizontal[2].Slave := 2.0, [5].Comas.Tete.Cam_Axe_Horizontal[3].Master := 31.0, [5].Comas.Tete.Cam_Axe_Horizontal[3].Slave := 27.0, [5].Comas.Tete.Cam_Axe_Horizontal[3].SegmentType := 1,
        [5].Comas.Tete.Cam_Axe_Horizontal[4].Master := 41.0, [5].Comas.Tete.Cam_Axe_Horizontal[4].Slave := 32.0, [5].Comas.Tete.Cam_Axe_Horizontal[5].Master := 46.0, [5].Comas.Tete.Cam_Axe_Horizontal[5].Slave := 32.0, [5].Comas.Tete.Cam_Axe_Horizontal[5].SegmentType := 1, [5].Comas.Tete.Cam_Axe_Horizontal[6].Master := 56.0, [5].Comas.Tete.Cam_Axe_Horizontal[6].Slave := 22.0, [5].Comas.Tete.Cam_Axe_Horizontal[6].SegmentType := 1, [5].Comas.Tete.Cam_Axe_Horizontal[7].Master := 70.0, [5].Comas.Tete.Cam_Axe_Vertical[1].Master := 1.0, [5].Comas.Tete.Cam_Axe_Vertical[2].Master := 6.0, [5].Comas.Tete.Cam_Axe_Vertical[3].Master := 21.0, [5].Comas.Tete.Cam_Axe_Vertical[3].SegmentType := 1, [5].Comas.Tete.Cam_Axe_Vertical[4].Master := 31.0, [5].Comas.Tete.Cam_Axe_Vertical[4].Slave := 10.0, [5].Comas.Tete.Cam_Axe_Vertical[5].Master := 51.0, [5].Comas.Tete.Cam_Axe_Vertical[5].Slave := 10.0, [5].Comas.Tete.Cam_Axe_Vertical[5].SegmentType := 1, [5].Comas.Tete.Cam_Axe_Vertical[6].Master := 66.0, [5].Comas.Tete.Cam_Axe_Vertical[7].Master := 70.0, [5].Comas.Tete.Longueur_Cam_Axe_H := 8, [5].Comas.Tete.Offset_Vertical_Gauche := 38.0, [5].Comas.Tete.Offset_Horizontal_Gauche := 95.0, [5].Comas.Tete.Cam_Axe_Horizontal_Pan.B.x := 1.0, [5].Comas.Tete.Cam_Axe_Horizontal_Pan.C.x := 5.0, [5].Comas.Tete.Cam_Axe_Horizontal_Pan.C.y := 2.0, [5].Comas.Tete.Cam_Axe_Horizontal_Pan.D.x := 25.0, [5].Comas.Tete.Cam_Axe_Horizontal_Pan.D.y := 25.0, [5].Comas.Tete.Cam_Axe_Horizontal_Pan.E.x := 10.0, [5].Comas.Tete.Cam_Axe_Horizontal_Pan.E.y := 5.0, [5].Comas.Tete.Cam_Axe_Horizontal_Pan.F.x := 5.0, [5].Comas.Tete.Cam_Axe_Horizontal_Pan.G.x := 10.0, [5].Comas.Tete.Cam_Axe_Horizontal_Pan.G.y := -10.0, [5].Comas.Tete.Cam_Axe_Vertical_Pan.K.x := -10.0, [5].Comas.Tete.Cam_Axe_Vertical_Pan.L.x := -10.0, [5].Comas.Tete.Cam_Axe_Vertical_Pan.L.y := 10.0, [5].Comas.Tete.Cam_Axe_Vertical_Pan.M.x := 5.0, [5].Comas.Tete.Cam_Axe_Vertical_Pan.M.y := 10.0, [5].Comas.Tete.Cam_Axe_Vertical_Pan.N.x := 10.0, [5].Comas.Tete.Offset_Vertical_Droit := 45.0, [5].Comas.Tete.Offset_Horizontal_Droit := 95.0, [5].Comas.Pompe.Start_Cam_Logique_Avance := -9.0, [5].Comas.Pompe.Stop_Cam_Logique_Avance := 16.0, [5].Comas.Pompe.Start_Cam_Logique_Recul := 21.0, [5].Comas.Pompe.Stop_Cam_Logique_Recul := 33.0, [5].Comas.Pompe.Consigne_Vitesse_Avance := 15.0, [5].Comas.Pompe.Consigne_Acc_Dec_Avance := 40.0, [5].Comas.Pompe.Consigne_Jerk_Avance := 100.0, [5].Comas.Pompe.Consigne_Vitesse_Recul := -15.0, [5].Comas.Pompe.Consigne_Acc_Dec_Recul := 40.0, [5].Comas.Pompe.Consigne_Jerk_Recul := 100.0, [5].Comas.Pompe.Points_Pan.O.x := -15.0, [5].Comas.Pompe.Points_Pan.Q.x := 25.0, [5].Comas.Pompe.Points_Pan.U.x := 12.0, [5].Comas.Pompe.Reserve_Bool1 := 1, [5].Comas.Rouleaux.Syncho_Pompe := 1, [5].Comas.Rouleaux.Consigne_Vitesse := 25.0, [5].Comas.Rouleaux.Consigne_Acc_Dec := 40.0, [5].Comas.Rouleaux.Consigne_Jerk := 100.0, [5].Comas.Coupe_Fil.Start_Cam_Logique_Virtuelle := 11.0,
        [5].Comas.Coupe_Fil.Stop_Cam_Logique_Virtuelle := 21.0, [5].Comas.Coupe_Fil.Consigne_Vitesse_Virtuelle := 200.0, [5].Comas.Coupe_Fil.Consigne_Acc_Dec_Virtuelle := 1000.0, [5].Comas.Coupe_Fil.Consigne_Jerk_Virtuelle := 50.0, [5].Comas.Coupe_Fil.Cam_Axe[0].SegmentType := 1, [5].Comas.Coupe_Fil.Cam_Axe[1].Master := 180.0, [5].Comas.Coupe_Fil.Cam_Axe[1].Slave := 90.0, [5].Comas.Coupe_Fil.Cam_Axe[2].Master := 360.0, [5].Comas.Coupe_Fil.Cam_Axe[2].Slave := 360.0, [5].Comas.Coupe_Fil.Cam_Axe[2].SegmentType := 1, [5].Comas.Coupe_Fil.Points_Pan.W.x := 30.0, [5].Comas.Consigne_Vitesse_Manu_mm := 4.0, [5].Comas.Consigne_Acc_Decc_Manu_mm := 10.0, [5].Comas.Consigne_Jerk_Manu := 100.0, [5].Comas.Activation_Cam_Auto := 1, [5].Comas.Distance_CPT_Presence_Produit := 520, [5].Comas.Consigne_Vitesse_Manu_Tour := 10.0, [5].Comas.Consigne_Acc_Decc_Manu_Tour := 10.0, [5].Comas.Mode_Decoreuse_Cam_Logique := 1, [5].Comas.Reserve_Real6 := 200.0, [6].Name := 'PALET CITRON 44', [6].Comas.Pas_Machine := 70, [6].Comas.Came_Maitre[1].Master := 70.0, [6].Comas.Came_Maitre[1].Slave := 70.0, [6].Comas.Longueur_Came_Maitre := 2, [6].Comas.Tete.Stop_Cam_Logique_Degagement := 10.0, [6].Comas.Tete.Position_Degagement_H := 50.0, [6].Comas.Tete.Position_Degagement_V := 35.0, [6].Comas.Tete.Hauteur_Tete := -3, [6].Comas.Tete.Cam_Axe_Horizontal[1].Master := 1.0, [6].Comas.Tete.Cam_Axe_Horizontal[1].SegmentType := 1, [6].Comas.Tete.Cam_Axe_Horizontal[2].Master := 6.0, [6].Comas.Tete.Cam_Axe_Horizontal[2].Slave := 2.0, [6].Comas.Tete.Cam_Axe_Horizontal[3].Master := 31.0, [6].Comas.Tete.Cam_Axe_Horizontal[3].Slave := 32.0, [6].Comas.Tete.Cam_Axe_Horizontal[3].SegmentType := 1, [6].Comas.Tete.Cam_Axe_Horizontal[4].Master := 41.0, [6].Comas.Tete.Cam_Axe_Horizontal[4].Slave := 42.0, [6].Comas.Tete.Cam_Axe_Horizontal[5].Master := 46.0, [6].Comas.Tete.Cam_Axe_Horizontal[5].Slave := 42.0, [6].Comas.Tete.Cam_Axe_Horizontal[5].SegmentType := 1, [6].Comas.Tete.Cam_Axe_Horizontal[6].Master := 56.0, [6].Comas.Tete.Cam_Axe_Horizontal[6].Slave := 32.0, [6].Comas.Tete.Cam_Axe_Horizontal[6].SegmentType := 1, [6].Comas.Tete.Cam_Axe_Horizontal[7].Master := 70.0, [6].Comas.Tete.Cam_Axe_Vertical[1].Master := 1.0, [6].Comas.Tete.Cam_Axe_Vertical[2].Master := 6.0, [6].Comas.Tete.Cam_Axe_Vertical[3].Master := 21.0, [6].Comas.Tete.Cam_Axe_Vertical[3].SegmentType := 1, [6].Comas.Tete.Cam_Axe_Vertical[4].Master := 31.0, [6].Comas.Tete.Cam_Axe_Vertical[4].Slave := 12.0, [6].Comas.Tete.Cam_Axe_Vertical[5].Master := 51.0, [6].Comas.Tete.Cam_Axe_Vertical[5].Slave := 5.0, [6].Comas.Tete.Cam_Axe_Vertical[5].SegmentType := 1, [6].Comas.Tete.Cam_Axe_Vertical[6].Master := 66.0, [6].Comas.Tete.Cam_Axe_Vertical[7].Master := 70.0, [6].Comas.Tete.Longueur_Cam_Axe_H := 8, [6].Comas.Tete.Offset_Vertical_Gauche := 38.0, [6].Comas.Tete.Offset_Horizontal_Gauche := 95.0, [6].Comas.Tete.Cam_Axe_Horizontal_Pan.B.x := 1.0,
